LIN {X 0,Y 320.619,Z 422.638,A -85,B 0,C 180,E1 -15590.529,E2 -15590.529} C_VEL
LIN {X 0,Y 322.237,Z 412.256,A -85,B 0,C 180,E1 -15591.593,E2 -15591.593} C_VEL
LIN {X 0,Y 323.7,Z 399.843,A -85,B 0,C 180,E1 -15592.581,E2 -15592.581} C_VEL
LIN {X 0,Y 325.026,Z 386.792,A -85,B 0,C 180,E1 -15593.324,E2 -15593.324} C_VEL
LIN {X 0,Y 325.91,Z 373.737,A -85,B 0,C 180,E1 -15593.805,E2 -15593.805} C_VEL
LIN {X 0,Y 327.738,Z 306.835,A -85,B 0,C 180,E1 -15595.344,E2 -15595.344} C_VEL
LIN {X 0,Y 324.36,Z 288.516,A -85,B 0,C 180,E1 -15596.163,E2 -15596.163} C_VEL
LIN {X 0,Y 321.852,Z 278.173,A -85,B 0,C 180,E1 -15596.706,E2 -15596.706} C_VEL
LIN {X 0,Y 317.141,Z 267.501,A -85,B 0,C 180,E1 -15597.567,E2 -15597.567} C_VEL
LIN {X 0,Y 315.127,Z 258.496,A -85,B 0,C 180,E1 -15600.525,E2 -15600.525} C_VEL
LIN {X 0,Y 312.559,Z 248.178,A -85,B 0,C 180,E1 -15604.298,E2 -15604.298} C_VEL
LIN {X 0,Y 312.491,Z 248.049,A -85,B 0,C 180,E1 -15608.074,E2 -15608.074} C_VEL
LIN {X 0,Y 312.492,Z 248.056,A -85,B 0,C 180,E1 -15610.706,E2 -15610.706} C_VEL
LIN {X 0,Y 312.454,Z 248.066,A -85,B 0,C 180,E1 -15614.206,E2 -15614.206} C_VEL
LIN {X 0,Y 312.457,Z 248.052,A -85,B 0,C 180,E1 -15617.921,E2 -15617.921} C_VEL
LIN {X 0,Y 312.477,Z 248.06,A -85,B 0,C 180,E1 -15621.92,E2 -15621.92} C_VEL
LIN {X 0,Y 312.531,Z 248.049,A -85,B 0,C 180,E1 -15624.216,E2 -15624.216} C_VEL
LIN {X 0,Y 312.501,Z 248.051,A -85,B 0,C 180,E1 -15627.329,E2 -15627.329} C_VEL
LIN {X 0,Y 312.504,Z 248.052,A -85,B 0,C 180,E1 -15631.287,E2 -15631.287} C_VEL
LIN {X 0,Y 312.519,Z 248.048,A -85,B 0,C 180,E1 -15634.701,E2 -15634.701} C_VEL
LIN {X 0,Y 312.534,Z 248.051,A -85,B 0,C 180,E1 -15637.521,E2 -15637.521} C_VEL
LIN {X 0,Y 312.561,Z 248.048,A -85,B 0,C 180,E1 -15641.647,E2 -15641.647} C_VEL
LIN {X 0,Y 312.678,Z 248.036,A -85,B 0,C 180,E1 -15645.681,E2 -15645.681} C_VEL
LIN {X 0,Y 312.675,Z 248.038,A -85,B 0,C 180,E1 -15649.636,E2 -15649.636} C_VEL
LIN {X 0,Y 312.791,Z 248.009,A -85,B 0,C 180,E1 -15652.248,E2 -15652.248} C_VEL
LIN {X 0,Y 312.678,Z 248.036,A -85,B 0,C 180,E1 -15654.837,E2 -15654.837} C_VEL
LIN {X 0,Y 312.965,Z 247.999,A -85,B 0,C 180,E1 -15658.708,E2 -15658.708} C_VEL
LIN {X 0,Y 312.889,Z 248.007,A -85,B 0,C 180,E1 -15662.57,E2 -15662.57} C_VEL
LIN {X 0,Y 312.822,Z 248.015,A -85,B 0,C 180,E1 -15666.445,E2 -15666.445} C_VEL
LIN {X 0,Y 312.732,Z 248.024,A -85,B 0,C 180,E1 -15669.045,E2 -15669.045} C_VEL
LIN {X 0,Y 312.614,Z 248.037,A -85,B 0,C 180,E1 -15672.986,E2 -15672.986} C_VEL
LIN {X 0,Y 312.6,Z 248.046,A -85,B 0,C 180,E1 -15675.646,E2 -15675.646} C_VEL
LIN {X 0,Y 312.537,Z 248.05,A -85,B 0,C 180,E1 -15679.707,E2 -15679.707} C_VEL
LIN {X 0,Y 312.501,Z 248.054,A -85,B 0,C 180,E1 -15682.776,E2 -15682.776} C_VEL
LIN {X 0,Y 312.576,Z 248.047,A -85,B 0,C 180,E1 -15685.931,E2 -15685.931} C_VEL
LIN {X 0,Y 312.51,Z 248.047,A -85,B 0,C 180,E1 -15689.647,E2 -15689.647} C_VEL
LIN {X 0,Y 312.489,Z 248.056,A -85,B 0,C 180,E1 -15693.685,E2 -15693.685} C_VEL
LIN {X 0,Y 312.544,Z 248.146,A -85,B 0,C 180,E1 -15696.984,E2 -15696.984} C_VEL
LIN {X 0,Y 314.824,Z 257.191,A -85,B 0,C 180,E1 -15700.336,E2 -15700.336} C_VEL
LIN {X 0,Y 315.609,Z 260.248,A -85,B 0,C 180,E1 -15701.299,E2 -15701.299} C_VEL
LIN {X 0,Y 322.41,Z 274.835,A -85,B 0,C 180,E1 -15702.504,E2 -15702.504} C_VEL
LIN {X 0,Y 325.404,Z 282.157,A -85,B 0,C 180,E1 -15703.019,E2 -15703.019} C_VEL
LIN {X 0,Y 328.126,Z 295.692,A -85,B 0,C 180,E1 -15703.648,E2 -15703.648} C_VEL
LIN {X 0,Y 325.864,Z 368.46,A -85,B 0,C 180,E1 -15705.321,E2 -15705.321} C_VEL
LIN {X 0,Y 324.969,Z 381.92,A -85,B 0,C 180,E1 -15705.887,E2 -15705.887} C_VEL
LIN {X 0,Y 323.783,Z 394.274,A -85,B 0,C 180,E1 -15706.654,E2 -15706.654} C_VEL
LIN {X 0,Y 322.337,Z 406.019,A -85,B 0,C 180,E1 -15707.647,E2 -15707.647} C_VEL
LIN {X 0,Y 320.627,Z 417.406,A -85,B 0,C 180,E1 -15708.887,E2 -15708.887} C_VEL
LIN {X 0,Y 318.918,Z 427.555,A -85,B 0,C 180,E1 -15710.28,E2 -15710.28} C_VEL
LIN {X 0,Y 317.347,Z 435.854,A -85,B 0,C 180,E1 -15711.68,E2 -15711.68} C_VEL
LIN {X 0,Y 315.656,Z 444.602,A -85,B 0,C 180,E1 -15713.507,E2 -15713.507} C_VEL
LIN {X 0,Y 314.073,Z 452.692,A -85,B 0,C 180,E1 -15715.638,E2 -15715.638} C_VEL
LIN {X 0,Y 313.006,Z 457.984,A -85,B 0,C 180,E1 -15717.395,E2 -15717.395} C_VEL
LIN {X 0,Y 312.043,Z 463.111,A -85,B 0,C 180,E1 -15719.555,E2 -15719.555} C_VEL
LIN {X 0,Y 311.358,Z 466.861,A -85,B 0,C 180,E1 -15721.707,E2 -15721.707} C_VEL
LIN {X 0,Y 310.953,Z 468.664,A -85,B 0,C 180,E1 -15723.129,E2 -15723.129} C_VEL
LIN {X 0,Y 310.645,Z 470.184,A -85,B 0,C 180,E1 -15724.801,E2 -15724.801} C_VEL
LIN {X 0,Y 310.353,Z 471.184,A -85,B 0,C 180,E1 -15727.361,E2 -15727.361} C_VEL
LIN {X 0,Y 310.339,Z 471.111,A -85,B 0,C 180,E1 -15728.758,E2 -15728.758} C_VEL
LIN {X 0,Y 310.34,Z 470.552,A -85,B 0,C 180,E1 -15730.144,E2 -15730.144} C_VEL
LIN {X 0,Y 310.435,Z 469.179,A -85,B 0,C 180,E1 -15731.938,E2 -15731.938} C_VEL
LIN {X 0,Y 310.741,Z 466.186,A -85,B 0,C 180,E1 -15734.254,E2 -15734.254} C_VEL
LIN {X 0,Y 311.132,Z 462.559,A -85,B 0,C 180,E1 -15736.21,E2 -15736.21} C_VEL
LIN {X 0,Y 311.583,Z 457.45,A -85,B 0,C 180,E1 -15738.29,E2 -15738.29} C_VEL
LIN {X 0,Y 312.253,Z 451.179,A -85,B 0,C 180,E1 -15740.284,E2 -15740.284} C_VEL
LIN {X 0,Y 313.202,Z 443.354,A -85,B 0,C 180,E1 -15742.265,E2 -15742.265} C_VEL
LIN {X 0,Y 314.209,Z 435.298,A -85,B 0,C 180,E1 -15743.903,E2 -15743.903} C_VEL
LIN {X 0,Y 315.35,Z 425.459,A -85,B 0,C 180,E1 -15745.528,E2 -15745.528} C_VEL
LIN {X 0,Y 316.667,Z 414.664,A -85,B 0,C 180,E1 -15746.955,E2 -15746.955} C_VEL
LIN {X 0,Y 317.737,Z 403.761,A -85,B 0,C 180,E1 -15748.101,E2 -15748.101} C_VEL
LIN {X 0,Y 318.799,Z 390.855,A -85,B 0,C 180,E1 -15749.134,E2 -15749.134} C_VEL
LIN {X 0,Y 319.644,Z 377.868,A -85,B 0,C 180,E1 -15749.884,E2 -15749.884} C_VEL
LIN {X 0,Y 320.152,Z 365.22,A -85,B 0,C 180,E1 -15750.356,E2 -15750.356} C_VEL
LIN {X 0,Y 321.67,Z 292.026,A -85,B 0,C 180,E1 -15752.026,E2 -15752.026} C_VEL
LIN {X 0,Y 317.467,Z 267.45,A -85,B 0,C 180,E1 -15752.877,E2 -15752.877} C_VEL
LIN {X 0,Y 315.024,Z 260.027,A -85,B 0,C 180,E1 -15753.263,E2 -15753.263} C_VEL
LIN {X 0,Y 312.877,Z 248.346,A -85,B 0,C 180,E1 -15756.937,E2 -15756.937} C_VEL
LIN {X 0,Y 312.847,Z 248.014,A -85,B 0,C 180,E1 -15757.424,E2 -15757.424} C_VEL
LIN {X 0,Y 312.633,Z 248.042,A -85,B 0,C 180,E1 -15761.675,E2 -15761.675} C_VEL
LIN {X 0,Y 312.665,Z 248.034,A -85,B 0,C 180,E1 -15764.891,E2 -15764.891} C_VEL
LIN {X 0,Y 312.575,Z 248.047,A -85,B 0,C 180,E1 -15769.229,E2 -15769.229} C_VEL
LIN {X 0,Y 312.485,Z 248.057,A -85,B 0,C 180,E1 -15772.781,E2 -15772.781} C_VEL
LIN {X 0,Y 312.48,Z 248.062,A -85,B 0,C 180,E1 -15775.905,E2 -15775.905} C_VEL
LIN {X 0,Y 312.466,Z 248.062,A -85,B 0,C 180,E1 -15779.66,E2 -15779.66} C_VEL
LIN {X 0,Y 312.492,Z 248.055,A -85,B 0,C 180,E1 -15783.694,E2 -15783.694} C_VEL
LIN {X 0,Y 312.484,Z 248.057,A -85,B 0,C 180,E1 -15787.393,E2 -15787.393} C_VEL
LIN {X 0,Y 312.417,Z 248.067,A -85,B 0,C 180,E1 -15790.723,E2 -15790.723} C_VEL
LIN {X 0,Y 312.429,Z 248.066,A -85,B 0,C 180,E1 -15794.216,E2 -15794.216} C_VEL
LIN {X 0,Y 312.407,Z 248.064,A -85,B 0,C 180,E1 -15795.376,E2 -15795.376} C_VEL
LIN {X 0,Y 311.764,Z 248.149,A -85,B 0,C 180,E1 -15796.452,E2 -15796.452} C_VEL
LIN {X 0,Y 308.895,Z 248.501,A -85,B 0,C 180,E1 -15798.203,E2 -15798.203} C_VEL
LIN {X 0,Y 306.465,Z 248.801,A -85,B 0,C 180,E1 -15799.623,E2 -15799.623} C_VEL
LIN {X 0,Y 305.454,Z 248.931,A -85,B 0,C 180,E1 -15800.724,E2 -15800.724} C_VEL
LIN {X 0,Y 305.389,Z 248.936,A -85,B 0,C 180,E1 -15801.096,E2 -15801.096} C_VEL
LIN {X 0,Y 305.447,Z 248.939,A -85,B 0,C 180,E1 -15804.893,E2 -15804.893} C_VEL
LIN {X 0,Y 305.43,Z 248.932,A -85,B 0,C 180,E1 -15808.365,E2 -15808.365} C_VEL
LIN {X 0,Y 305.442,Z 248.928,A -85,B 0,C 180,E1 -15811.113,E2 -15811.113} C_VEL
LIN {X 0,Y 305.471,Z 248.93,A -85,B 0,C 180,E1 -15814.086,E2 -15814.086} C_VEL
LIN {X 0,Y 305.457,Z 248.932,A -85,B 0,C 180,E1 -15818.406,E2 -15818.406} C_VEL
LIN {X 0,Y 305.533,Z 248.912,A -85,B 0,C 180,E1 -15822.607,E2 -15822.607} C_VEL
LIN {X 0,Y 305.626,Z 248.906,A -85,B 0,C 180,E1 -15825.354,E2 -15825.354} C_VEL
LIN {X 0,Y 305.625,Z 248.913,A -85,B 0,C 180,E1 -15829.405,E2 -15829.405} C_VEL
LIN {X 0,Y 305.75,Z 248.898,A -85,B 0,C 180,E1 -15832.078,E2 -15832.078} C_VEL
LIN {X 0,Y 305.661,Z 248.9,A -85,B 0,C 180,E1 -15834.728,E2 -15834.728} C_VEL
LIN {X 0,Y 305.942,Z 248.868,A -85,B 0,C 180,E1 -15838.689,E2 -15838.689} C_VEL
LIN {X 0,Y 305.952,Z 248.87,A -85,B 0,C 180,E1 -15841.321,E2 -15841.321} C_VEL
LIN {X 0,Y 305.794,Z 248.889,A -85,B 0,C 180,E1 -15846.604,E2 -15846.604} C_VEL
LIN {X 0,Y 305.696,Z 248.892,A -85,B 0,C 180,E1 -15849.266,E2 -15849.266} C_VEL
LIN {X 0,Y 305.6,Z 248.915,A -85,B 0,C 180,E1 -15853.3,E2 -15853.3} C_VEL
LIN {X 0,Y 305.565,Z 248.92,A -85,B 0,C 180,E1 -15856.026,E2 -15856.026} C_VEL
LIN {X 0,Y 305.499,Z 248.921,A -85,B 0,C 180,E1 -15860.191,E2 -15860.191} C_VEL
LIN {X 0,Y 305.49,Z 248.93,A -85,B 0,C 180,E1 -15864.467,E2 -15864.467} C_VEL
LIN {X 0,Y 305.471,Z 248.931,A -85,B 0,C 180,E1 -15867.401,E2 -15867.401} C_VEL
LIN {X 0,Y 305.447,Z 248.929,A -85,B 0,C 180,E1 -15870.415,E2 -15870.415} C_VEL
LIN {X 0,Y 305.483,Z 248.93,A -85,B 0,C 180,E1 -15874.08,E2 -15874.08} C_VEL
LIN {X 0,Y 305.47,Z 248.928,A -85,B 0,C 180,E1 -15876.745,E2 -15876.745} C_VEL
LIN {X 0,Y 305.427,Z 248.937,A -85,B 0,C 180,E1 -15880.591,E2 -15880.591} C_VEL
LIN {X 0,Y 305.438,Z 248.938,A -85,B 0,C 180,E1 -15883.658,E2 -15883.658} C_VEL
LIN {X 0,Y 305.452,Z 248.935,A -85,B 0,C 180,E1 -15887.42,E2 -15887.42} C_VEL
LIN {X 0,Y 305.46,Z 248.933,A -85,B 0,C 180,E1 -15891.593,E2 -15891.593} C_VEL
LIN {X 0,Y 305.48,Z 248.929,A -85,B 0,C 180,E1 -15894.887,E2 -15894.887} C_VEL
LIN {X 0,Y 305.496,Z 248.932,A -85,B 0,C 180,E1 -15899.21,E2 -15899.21} C_VEL
LIN {X 0,Y 305.545,Z 249.228,A -85,B 0,C 180,E1 -15899.598,E2 -15899.598} C_VEL
LIN {X 0,Y 307.891,Z 260.415,A -85,B 0,C 180,E1 -15903.16,E2 -15903.16} C_VEL
LIN {X 0,Y 309.119,Z 267.787,A -85,B 0,C 180,E1 -15905.355,E2 -15905.355} C_VEL
LIN {X 0,Y 309.705,Z 271.988,A -85,B 0,C 180,E1 -15905.575,E2 -15905.575} C_VEL
LIN {X 0,Y 314.832,Z 306.06,A -85,B 0,C 180,E1 -15906.74,E2 -15906.74} C_VEL
LIN {X 0,Y 313.293,Z 375.551,A -85,B 0,C 180,E1 -15908.36,E2 -15908.36} C_VEL
LIN {X 0,Y 312.561,Z 388.819,A -85,B 0,C 180,E1 -15908.912,E2 -15908.912} C_VEL
LIN {X 0,Y 311.622,Z 401.603,A -85,B 0,C 180,E1 -15909.709,E2 -15909.709} C_VEL
LIN {X 0,Y 310.524,Z 412.959,A -85,B 0,C 180,E1 -15910.668,E2 -15910.668} C_VEL
LIN {X 0,Y 309.219,Z 424.684,A -85,B 0,C 180,E1 -15911.959,E2 -15911.959} C_VEL
LIN {X 0,Y 308.095,Z 434.783,A -85,B 0,C 180,E1 -15913.359,E2 -15913.359} C_VEL
LIN {X 0,Y 306.849,Z 444.708,A -85,B 0,C 180,E1 -15915.066,E2 -15915.066} C_VEL
LIN {X 0,Y 305.693,Z 453.833,A -85,B 0,C 180,E1 -15917.045,E2 -15917.045} C_VEL
LIN {X 0,Y 304.827,Z 461.173,A -85,B 0,C 180,E1 -15919.033,E2 -15919.033} C_VEL
LIN {X 0,Y 304.287,Z 466.122,A -85,B 0,C 180,E1 -15920.694,E2 -15920.694} C_VEL
LIN {X 0,Y 303.861,Z 470.917,A -85,B 0,C 180,E1 -15922.69,E2 -15922.69} C_VEL
LIN {X 0,Y 303.653,Z 474.574,A -85,B 0,C 180,E1 -15924.686,E2 -15924.686} C_VEL
LIN {X 0,Y 303.595,Z 476.458,A -85,B 0,C 180,E1 -15926.016,E2 -15926.016} C_VEL
LIN {X 0,Y 303.587,Z 477.869,A -85,B 0,C 180,E1 -15927.344,E2 -15927.344} C_VEL
LIN {X 0,Y 303.535,Z 478.867,A -85,B 0,C 180,E1 -15928.671,E2 -15928.671} C_VEL
LIN {X 0,Y 303.542,Z 479.476,A -85,B 0,C 180,E1 -15929.998,E2 -15929.998} C_VEL
LIN {X 0,Y 303.535,Z 479.694,A -85,B 0,C 180,E1 -15931.325,E2 -15931.325} C_VEL
LIN {X 0,Y 303.589,Z 479.483,A -85,B 0,C 180,E1 -15932.652,E2 -15932.652} C_VEL
LIN {X 0,Y 303.699,Z 477.887,A -85,B 0,C 180,E1 -15935.309,E2 -15935.309} C_VEL
LIN {X 0,Y 303.851,Z 476.507,A -85,B 0,C 180,E1 -15936.639,E2 -15936.639} C_VEL
LIN {X 0,Y 304.3,Z 473.604,A -85,B 0,C 180,E1 -15938.632,E2 -15938.632} C_VEL
LIN {X 0,Y 305,Z 469.69,A -85,B 0,C 180,E1 -15940.621,E2 -15940.621} C_VEL
LIN {X 0,Y 306.006,Z 464.664,A -85,B 0,C 180,E1 -15942.6,E2 -15942.6} C_VEL
LIN {X 0,Y 307.33,Z 458.369,A -85,B 0,C 180,E1 -15944.567,E2 -15944.567} C_VEL
LIN {X 0,Y 309.055,Z 450.506,A -85,B 0,C 180,E1 -15946.512,E2 -15946.512} C_VEL
LIN {X 0,Y 310.649,Z 441.952,A -85,B 0,C 180,E1 -15948.233,E2 -15948.233} C_VEL
LIN {X 0,Y 312.581,Z 431.757,A -85,B 0,C 180,E1 -15949.879,E2 -15949.879} C_VEL
LIN {X 0,Y 314.528,Z 420.616,A -85,B 0,C 180,E1 -15951.288,E2 -15951.288} C_VEL
LIN {X 0,Y 316.212,Z 409.737,A -85,B 0,C 180,E1 -15952.369,E2 -15952.369} C_VEL
LIN {X 0,Y 317.624,Z 397.768,A -85,B 0,C 180,E1 -15953.296,E2 -15953.296} C_VEL
LIN {X 0,Y 318.852,Z 385.459,A -85,B 0,C 180,E1 -15953.976,E2 -15953.976} C_VEL
LIN {X 0,Y 319.721,Z 372.89,A -85,B 0,C 180,E1 -15954.424,E2 -15954.424} C_VEL
LIN {X 0,Y 321.568,Z 307.683,A -85,B 0,C 180,E1 -15955.957,E2 -15955.957} C_VEL
LIN {X 0,Y 318.048,Z 288.778,A -85,B 0,C 180,E1 -15956.845,E2 -15956.845} C_VEL
LIN {X 0,Y 316.233,Z 281.362,A -85,B 0,C 180,E1 -15957.25,E2 -15957.25} C_VEL
LIN {X 0,Y 309.98,Z 267.54,A -85,B 0,C 180,E1 -15958.398,E2 -15958.398} C_VEL
LIN {X 0,Y 309.111,Z 263.636,A -85,B 0,C 180,E1 -15959.635,E2 -15959.635} C_VEL
LIN {X 0,Y 307.104,Z 255.27,A -85,B 0,C 180,E1 -15962.637,E2 -15962.637} C_VEL
LIN {X 0,Y 305.514,Z 249.002,A -85,B 0,C 180,E1 -15965.103,E2 -15965.103} C_VEL
LIN {X 0,Y 305.431,Z 248.928,A -85,B 0,C 180,E1 -15968.519,E2 -15968.519} C_VEL
LIN {X 0,Y 305.431,Z 248.924,A -85,B 0,C 180,E1 -15971.855,E2 -15971.855} C_VEL
LIN {X 0,Y 305.402,Z 248.93,A -85,B 0,C 180,E1 -15975.507,E2 -15975.507} C_VEL
LIN {X 0,Y 305.414,Z 248.932,A -85,B 0,C 180,E1 -15978.134,E2 -15978.134} C_VEL
LIN {X 0,Y 305.442,Z 248.936,A -85,B 0,C 180,E1 -15981.588,E2 -15981.588} C_VEL
LIN {X 0,Y 305.462,Z 248.935,A -85,B 0,C 180,E1 -15984.882,E2 -15984.882} C_VEL
LIN {X 0,Y 305.441,Z 248.935,A -85,B 0,C 180,E1 -15988.354,E2 -15988.354} C_VEL
LIN {X 0,Y 305.473,Z 248.927,A -85,B 0,C 180,E1 -15991.104,E2 -15991.104} C_VEL
LIN {X 0,Y 305.478,Z 248.928,A -85,B 0,C 180,E1 -15994.075,E2 -15994.075} C_VEL
LIN {X 0,Y 305.458,Z 248.928,A -85,B 0,C 180,E1 -15998.395,E2 -15998.395} C_VEL
LIN {X 0,Y 305.529,Z 248.92,A -85,B 0,C 180,E1 -16002.596,E2 -16002.596} C_VEL
LIN {X 0,Y 305.619,Z 248.917,A -85,B 0,C 180,E1 -16005.343,E2 -16005.343} C_VEL
LIN {X 0,Y 305.614,Z 248.915,A -85,B 0,C 180,E1 -16009.394,E2 -16009.394} C_VEL
LIN {X 0,Y 305.74,Z 248.888,A -85,B 0,C 180,E1 -16012.068,E2 -16012.068} C_VEL
LIN {X 0,Y 305.649,Z 248.911,A -85,B 0,C 180,E1 -16014.718,E2 -16014.718} C_VEL
LIN {X 0,Y 305.931,Z 248.875,A -85,B 0,C 180,E1 -16018.679,E2 -16018.679} C_VEL
LIN {X 0,Y 305.92,Z 248.869,A -85,B 0,C 180,E1 -16021.311,E2 -16021.311} C_VEL
LIN {X 0,Y 305.641,Z 248.905,A -85,B 0,C 180,E1 -16025.272,E2 -16025.272} C_VEL
LIN {X 0,Y 305.728,Z 248.902,A -85,B 0,C 180,E1 -16027.922,E2 -16027.922} C_VEL
LIN {X 0,Y 305.579,Z 248.92,A -85,B 0,C 180,E1 -16031.94,E2 -16031.94} C_VEL
LIN {X 0,Y 305.588,Z 248.919,A -85,B 0,C 180,E1 -16035.009,E2 -16035.009} C_VEL
LIN {X 0,Y 305.519,Z 248.924,A -85,B 0,C 180,E1 -16039.422,E2 -16039.422} C_VEL
LIN {X 0,Y 305.461,Z 248.932,A -85,B 0,C 180,E1 -16043.035,E2 -16043.035} C_VEL
LIN {X 0,Y 305.52,Z 248.929,A -85,B 0,C 180,E1 -16046.222,E2 -16046.222} C_VEL
LIN {X 0,Y 305.46,Z 248.92,A -85,B 0,C 180,E1 -16049.043,E2 -16049.043} C_VEL
LIN {X 0,Y 305.413,Z 248.932,A -85,B 0,C 180,E1 -16051.948,E2 -16051.948} C_VEL
LIN {X 0,Y 305.484,Z 249.005,A -85,B 0,C 180,E1 -16056.206,E2 -16056.206} C_VEL
LIN {X 0,Y 307.819,Z 258.157,A -85,B 0,C 180,E1 -16059.73,E2 -16059.73} C_VEL
LIN {X 0,Y 308.403,Z 260.428,A -85,B 0,C 180,E1 -16060.439,E2 -16060.439} C_VEL
LIN {X 0,Y 314.332,Z 272.513,A -85,B 0,C 180,E1 -16061.526,E2 -16061.526} C_VEL
LIN {X 0,Y 319.535,Z 284.486,A -85,B 0,C 180,E1 -16062.442,E2 -16062.442} C_VEL
LIN {X 0,Y 321.983,Z 297,A -85,B 0,C 180,E1 -16063.042,E2 -16063.042} C_VEL
LIN {X 0,Y 319.664,Z 368.312,A -85,B 0,C 180,E1 -16064.714,E2 -16064.714} C_VEL
LIN {X 0,Y 318.791,Z 381.04,A -85,B 0,C 180,E1 -16065.248,E2 -16065.248} C_VEL
LIN {X 0,Y 317.528,Z 393.61,A -85,B 0,C 180,E1 -16066.021,E2 -16066.021} C_VEL
LIN {X 0,Y 316.09,Z 405.087,A -85,B 0,C 180,E1 -16066.983,E2 -16066.983} C_VEL
LIN {X 0,Y 314.228,Z 417.05,A -85,B 0,C 180,E1 -16068.291,E2 -16068.291} C_VEL
LIN {X 0,Y 312.416,Z 427.335,A -85,B 0,C 180,E1 -16069.717,E2 -16069.717} C_VEL
LIN {X 0,Y 310.769,Z 435.634,A -85,B 0,C 180,E1 -16071.133,E2 -16071.133} C_VEL
LIN {X 0,Y 308.931,Z 444.73,A -85,B 0,C 180,E1 -16073.062,E2 -16073.062} C_VEL
LIN {X 0,Y 307.298,Z 452.462,A -85,B 0,C 180,E1 -16075.13,E2 -16075.13} C_VEL
LIN {X 0,Y 305.951,Z 458.903,A -85,B 0,C 180,E1 -16077.331,E2 -16077.331} C_VEL
LIN {X 0,Y 304.951,Z 463.792,A -85,B 0,C 180,E1 -16079.537,E2 -16079.537} C_VEL
LIN {X 0,Y 304.382,Z 466.801,A -85,B 0,C 180,E1 -16081.315,E2 -16081.315} C_VEL
LIN {X 0,Y 303.707,Z 469.752,A -85,B 0,C 180,E1 -16083.92,E2 -16083.92} C_VEL
LIN {X 0,Y 303.474,Z 470.741,A -85,B 0,C 180,E1 -16085.366,E2 -16085.366} C_VEL
LIN {X 0,Y 303.261,Z 471.3,A -85,B 0,C 180,E1 -16087.951,E2 -16087.951} C_VEL
LIN {X 0,Y 303.22,Z 470.862,A -85,B 0,C 180,E1 -16089.658,E2 -16089.658} C_VEL
LIN {X 0,Y 303.319,Z 469.386,A -85,B 0,C 180,E1 -16091.779,E2 -16091.779} C_VEL
LIN {X 0,Y 303.686,Z 465.807,A -85,B 0,C 180,E1 -16094.568,E2 -16094.568} C_VEL
LIN {X 0,Y 304.108,Z 461.865,A -85,B 0,C 180,E1 -16096.64,E2 -16096.64} C_VEL
LIN {X 0,Y 304.622,Z 456.742,A -85,B 0,C 180,E1 -16098.693,E2 -16098.693} C_VEL
LIN {X 0,Y 305.369,Z 450.28,A -85,B 0,C 180,E1 -16100.731,E2 -16100.731} C_VEL
LIN {X 0,Y 306.38,Z 442.144,A -85,B 0,C 180,E1 -16102.754,E2 -16102.754} C_VEL
LIN {X 0,Y 307.427,Z 433.829,A -85,B 0,C 180,E1 -16104.427,E2 -16104.427} C_VEL
LIN {X 0,Y 308.7,Z 423.659,A -85,B 0,C 180,E1 -16106.086,E2 -16106.086} C_VEL
LIN {X 0,Y 309.898,Z 413.559,A -85,B 0,C 180,E1 -16107.402,E2 -16107.402} C_VEL
LIN {X 0,Y 311.012,Z 402.562,A -85,B 0,C 180,E1 -16108.545,E2 -16108.545} C_VEL
LIN {X 0,Y 312.019,Z 390.453,A -85,B 0,C 180,E1 -16109.518,E2 -16109.518} C_VEL
LIN {X 0,Y 312.834,Z 378.084,A -85,B 0,C 180,E1 -16110.243,E2 -16110.243} C_VEL
LIN {X 0,Y 313.35,Z 365.555,A -85,B 0,C 180,E1 -16110.725,E2 -16110.725} C_VEL
LIN {X 0,Y 314.878,Z 292.515,A -85,B 0,C 180,E1 -16112.43,E2 -16112.43} C_VEL
LIN {X 0,Y 311.028,Z 269.782,A -85,B 0,C 180,E1 -16113.233,E2 -16113.233} C_VEL
LIN {X 0,Y 307.869,Z 260.473,A -85,B 0,C 180,E1 -16113.707,E2 -16113.707} C_VEL
LIN {X 0,Y 307.408,Z 258.332,A -85,B 0,C 180,E1 -16114.263,E2 -16114.263} C_VEL
LIN {X 0,Y 305.847,Z 249.195,A -85,B 0,C 180,E1 -16117.263,E2 -16117.263} C_VEL
LIN {X 0,Y 305.759,Z 248.899,A -85,B 0,C 180,E1 -16117.929,E2 -16117.929} C_VEL
LIN {X 0,Y 305.567,Z 248.921,A -85,B 0,C 180,E1 -16121.948,E2 -16121.948} C_VEL
LIN {X 0,Y 305.603,Z 248.915,A -85,B 0,C 180,E1 -16125.038,E2 -16125.038} C_VEL
LIN {X 0,Y 305.545,Z 248.921,A -85,B 0,C 180,E1 -16128.787,E2 -16128.787} C_VEL
LIN {X 0,Y 305.439,Z 248.935,A -85,B 0,C 180,E1 -16133.037,E2 -16133.037} C_VEL
LIN {X 0,Y 305.424,Z 248.939,A -85,B 0,C 180,E1 -16136.196,E2 -16136.196} C_VEL
LIN {X 0,Y 305.418,Z 248.939,A -85,B 0,C 180,E1 -16139.038,E2 -16139.038} C_VEL
LIN {X 0,Y 305.407,Z 248.941,A -85,B 0,C 180,E1 -16141.958,E2 -16141.958} C_VEL
LIN {X 0,Y 305.434,Z 248.936,A -85,B 0,C 180,E1 -16145.119,E2 -16145.119} C_VEL
LIN {X 0,Y 305.41,Z 248.939,A -85,B 0,C 180,E1 -16148.53,E2 -16148.53} C_VEL
LIN {X 0,Y 305.412,Z 248.942,A -85,B 0,C 180,E1 -16152.587,E2 -16152.587} C_VEL
LIN {X 0,Y 305.401,Z 248.941,A -85,B 0,C 180,E1 -16156.35,E2 -16156.35} C_VEL
LIN {X 0,Y 305.393,Z 248.934,A -85,B 0,C 180,E1 -16159.891,E2 -16159.891} C_VEL
LIN {X 0,Y 305.389,Z 248.936,A -85,B 0,C 180,E1 -16161.096,E2 -16161.096} C_VEL
LIN {X 0,Y 304.761,Z 249.02,A -85,B 0,C 180,E1 -16162.197,E2 -16162.197} C_VEL
LIN {X 0,Y 301.896,Z 249.376,A -85,B 0,C 180,E1 -16163.987,E2 -16163.987} C_VEL
LIN {X 0,Y 299.458,Z 249.681,A -85,B 0,C 180,E1 -16165.44,E2 -16165.44} C_VEL
LIN {X 0,Y 298.435,Z 249.808,A -85,B 0,C 180,E1 -16166.566,E2 -16166.566} C_VEL
LIN {X 0,Y 298.367,Z 249.813,A -85,B 0,C 180,E1 -16166.948,E2 -16166.948} C_VEL
LIN {X 0,Y 298.354,Z 249.806,A -85,B 0,C 180,E1 -16170.645,E2 -16170.645} C_VEL
LIN {X 0,Y 298.41,Z 249.811,A -85,B 0,C 180,E1 -16174.924,E2 -16174.924} C_VEL
LIN {X 0,Y 298.388,Z 249.814,A -85,B 0,C 180,E1 -16177.868,E2 -16177.868} C_VEL
LIN {X 0,Y 298.46,Z 249.799,A -85,B 0,C 180,E1 -16180.758,E2 -16180.758} C_VEL
LIN {X 0,Y 298.586,Z 249.78,A -85,B 0,C 180,E1 -16185,E2 -16185} C_VEL
LIN {X 0,Y 298.584,Z 249.789,A -85,B 0,C 180,E1 -16189.152,E2 -16189.152} C_VEL
LIN {X 0,Y 298.701,Z 249.777,A -85,B 0,C 180,E1 -16191.89,E2 -16191.89} C_VEL
LIN {X 0,Y 298.631,Z 249.775,A -85,B 0,C 180,E1 -16194.604,E2 -16194.604} C_VEL
LIN {X 0,Y 298.91,Z 249.744,A -85,B 0,C 180,E1 -16198.658,E2 -16198.658} C_VEL
LIN {X 0,Y 298.918,Z 249.746,A -85,B 0,C 180,E1 -16201.352,E2 -16201.352} C_VEL
LIN {X 0,Y 298.743,Z 249.766,A -85,B 0,C 180,E1 -16206.76,E2 -16206.76} C_VEL
LIN {X 0,Y 298.629,Z 249.77,A -85,B 0,C 180,E1 -16209.487,E2 -16209.487} C_VEL
LIN {X 0,Y 298.559,Z 249.791,A -85,B 0,C 180,E1 -16213.62,E2 -16213.62} C_VEL
LIN {X 0,Y 298.499,Z 249.803,A -85,B 0,C 180,E1 -16216.416,E2 -16216.416} C_VEL
LIN {X 0,Y 298.461,Z 249.797,A -85,B 0,C 180,E1 -16219.622,E2 -16219.622} C_VEL
LIN {X 0,Y 298.437,Z 249.807,A -85,B 0,C 180,E1 -16223.604,E2 -16223.604} C_VEL
LIN {X 0,Y 298.424,Z 249.811,A -85,B 0,C 180,E1 -16226.585,E2 -16226.585} C_VEL
LIN {X 0,Y 298.41,Z 249.806,A -85,B 0,C 180,E1 -16229.647,E2 -16229.647} C_VEL
LIN {X 0,Y 298.411,Z 249.812,A -85,B 0,C 180,E1 -16232.803,E2 -16232.803} C_VEL
LIN {X 0,Y 298.444,Z 249.803,A -85,B 0,C 180,E1 -16236.804,E2 -16236.804} C_VEL
LIN {X 0,Y 298.365,Z 249.82,A -85,B 0,C 180,E1 -16241.27,E2 -16241.27} C_VEL
LIN {X 0,Y 298.374,Z 249.817,A -85,B 0,C 180,E1 -16245.036,E2 -16245.036} C_VEL
LIN {X 0,Y 298.365,Z 249.817,A -85,B 0,C 180,E1 -16248.923,E2 -16248.923} C_VEL
LIN {X 0,Y 298.405,Z 249.811,A -85,B 0,C 180,E1 -16252.238,E2 -16252.238} C_VEL
LIN {X 0,Y 298.426,Z 249.809,A -85,B 0,C 180,E1 -16255.581,E2 -16255.581} C_VEL
LIN {X 0,Y 298.482,Z 249.977,A -85,B 0,C 180,E1 -16259.193,E2 -16259.193} C_VEL
LIN {X 0,Y 300.666,Z 260.544,A -85,B 0,C 180,E1 -16262.66,E2 -16262.66} C_VEL
LIN {X 0,Y 301.982,Z 267.843,A -85,B 0,C 180,E1 -16264.888,E2 -16264.888} C_VEL
LIN {X 0,Y 302.909,Z 271.921,A -85,B 0,C 180,E1 -16265.107,E2 -16265.107} C_VEL
LIN {X 0,Y 308.143,Z 307.18,A -85,B 0,C 180,E1 -16266.344,E2 -16266.344} C_VEL
LIN {X 0,Y 306.506,Z 375.971,A -85,B 0,C 180,E1 -16267.989,E2 -16267.989} C_VEL
LIN {X 0,Y 305.707,Z 389.831,A -85,B 0,C 180,E1 -16268.593,E2 -16268.593} C_VEL
LIN {X 0,Y 304.752,Z 402.31,A -85,B 0,C 180,E1 -16269.408,E2 -16269.408} C_VEL
LIN {X 0,Y 303.61,Z 413.44,A -85,B 0,C 180,E1 -16270.386,E2 -16270.386} C_VEL
LIN {X 0,Y 302.268,Z 425.059,A -85,B 0,C 180,E1 -16271.704,E2 -16271.704} C_VEL
LIN {X 0,Y 301.125,Z 435.026,A -85,B 0,C 180,E1 -16273.129,E2 -16273.129} C_VEL
LIN {X 0,Y 299.968,Z 444.073,A -85,B 0,C 180,E1 -16274.716,E2 -16274.716} C_VEL
LIN {X 0,Y 298.744,Z 453.301,A -85,B 0,C 180,E1 -16276.738,E2 -16276.738} C_VEL
LIN {X 0,Y 297.819,Z 460.717,A -85,B 0,C 180,E1 -16278.772,E2 -16278.772} C_VEL
LIN {X 0,Y 297.258,Z 465.735,A -85,B 0,C 180,E1 -16280.472,E2 -16280.472} C_VEL
LIN {X 0,Y 296.807,Z 470.592,A -85,B 0,C 180,E1 -16282.515,E2 -16282.515} C_VEL
LIN {X 0,Y 296.568,Z 474.306,A -85,B 0,C 180,E1 -16284.559,E2 -16284.559} C_VEL
LIN {X 0,Y 296.498,Z 476.22,A -85,B 0,C 180,E1 -16285.92,E2 -16285.92} C_VEL
LIN {X 0,Y 296.492,Z 477.681,A -85,B 0,C 180,E1 -16287.281,E2 -16287.281} C_VEL
LIN {X 0,Y 296.457,Z 478.706,A -85,B 0,C 180,E1 -16288.639,E2 -16288.639} C_VEL
LIN {X 0,Y 296.46,Z 479.34,A -85,B 0,C 180,E1 -16289.998,E2 -16289.998} C_VEL
LIN {X 0,Y 296.457,Z 479.586,A -85,B 0,C 180,E1 -16291.356,E2 -16291.356} C_VEL
LIN {X 0,Y 296.495,Z 479.421,A -85,B 0,C 180,E1 -16292.715,E2 -16292.715} C_VEL
LIN {X 0,Y 296.614,Z 477.876,A -85,B 0,C 180,E1 -16295.436,E2 -16295.436} C_VEL
LIN {X 0,Y 296.774,Z 476.522,A -85,B 0,C 180,E1 -16296.798,E2 -16296.798} C_VEL
LIN {X 0,Y 297.283,Z 473.671,A -85,B 0,C 180,E1 -16298.837,E2 -16298.837} C_VEL
LIN {X 0,Y 298.009,Z 469.812,A -85,B 0,C 180,E1 -16300.873,E2 -16300.873} C_VEL
LIN {X 0,Y 299.061,Z 464.845,A -85,B 0,C 180,E1 -16302.898,E2 -16302.898} C_VEL
LIN {X 0,Y 300.465,Z 458.623,A -85,B 0,C 180,E1 -16304.907,E2 -16304.907} C_VEL
LIN {X 0,Y 302.274,Z 450.863,A -85,B 0,C 180,E1 -16306.893,E2 -16306.893} C_VEL
LIN {X 0,Y 303.891,Z 442.669,A -85,B 0,C 180,E1 -16308.601,E2 -16308.601} C_VEL
LIN {X 0,Y 305.755,Z 433.401,A -85,B 0,C 180,E1 -16310.166,E2 -16310.166} C_VEL
LIN {X 0,Y 307.705,Z 422.794,A -85,B 0,C 180,E1 -16311.608,E2 -16311.608} C_VEL
LIN {X 0,Y 309.462,Z 412.535,A -85,B 0,C 180,E1 -16312.708,E2 -16312.708} C_VEL
LIN {X 0,Y 311.054,Z 400.329,A -85,B 0,C 180,E1 -16313.73,E2 -16313.73} C_VEL
LIN {X 0,Y 312.475,Z 387.547,A -85,B 0,C 180,E1 -16314.497,E2 -16314.497} C_VEL
LIN {X 0,Y 313.411,Z 375.296,A -85,B 0,C 180,E1 -16314.994,E2 -16314.994} C_VEL
LIN {X 0,Y 315.544,Z 309.217,A -85,B 0,C 180,E1 -16316.574,E2 -16316.574} C_VEL
LIN {X 0,Y 312.147,Z 290.747,A -85,B 0,C 180,E1 -16317.466,E2 -16317.466} C_VEL
LIN {X 0,Y 310.492,Z 284.171,A -85,B 0,C 180,E1 -16317.843,E2 -16317.843} C_VEL
LIN {X 0,Y 304.299,Z 270.733,A -85,B 0,C 180,E1 -16318.989,E2 -16318.989} C_VEL
LIN {X 0,Y 302.698,Z 267.125,A -85,B 0,C 180,E1 -16319.367,E2 -16319.367} C_VEL
LIN {X 0,Y 300.526,Z 257.979,A -85,B 0,C 180,E1 -16322.654,E2 -16322.654} C_VEL
LIN {X 0,Y 298.485,Z 249.854,A -85,B 0,C 180,E1 -16325.933,E2 -16325.933} C_VEL
LIN {X 0,Y 298.401,Z 249.811,A -85,B 0,C 180,E1 -16329.484,E2 -16329.484} C_VEL
LIN {X 0,Y 298.404,Z 249.804,A -85,B 0,C 180,E1 -16333.099,E2 -16333.099} C_VEL
LIN {X 0,Y 298.373,Z 249.797,A -85,B 0,C 180,E1 -16336.91,E2 -16336.91} C_VEL
LIN {X 0,Y 298.386,Z 249.812,A -85,B 0,C 180,E1 -16341.006,E2 -16341.006} C_VEL
LIN {X 0,Y 298.405,Z 249.808,A -85,B 0,C 180,E1 -16343.923,E2 -16343.923} C_VEL
LIN {X 0,Y 298.392,Z 249.808,A -85,B 0,C 180,E1 -16347.195,E2 -16347.195} C_VEL
LIN {X 0,Y 298.4,Z 249.808,A -85,B 0,C 180,E1 -16350.62,E2 -16350.62} C_VEL
LIN {X 0,Y 298.419,Z 249.804,A -85,B 0,C 180,E1 -16354.913,E2 -16354.913} C_VEL
LIN {X 0,Y 298.413,Z 249.804,A -85,B 0,C 180,E1 -16359.308,E2 -16359.308} C_VEL
LIN {X 0,Y 298.46,Z 249.804,A -85,B 0,C 180,E1 -16362.17,E2 -16362.17} C_VEL
LIN {X 0,Y 298.579,Z 249.791,A -85,B 0,C 180,E1 -16364.989,E2 -16364.989} C_VEL
LIN {X 0,Y 298.573,Z 249.788,A -85,B 0,C 180,E1 -16369.141,E2 -16369.141} C_VEL
LIN {X 0,Y 298.691,Z 249.767,A -85,B 0,C 180,E1 -16371.879,E2 -16371.879} C_VEL
LIN {X 0,Y 298.619,Z 249.786,A -85,B 0,C 180,E1 -16374.593,E2 -16374.593} C_VEL
LIN {X 0,Y 298.898,Z 249.751,A -85,B 0,C 180,E1 -16378.648,E2 -16378.648} C_VEL
LIN {X 0,Y 298.888,Z 249.744,A -85,B 0,C 180,E1 -16381.342,E2 -16381.342} C_VEL
LIN {X 0,Y 298.716,Z 249.773,A -85,B 0,C 180,E1 -16386.75,E2 -16386.75} C_VEL
LIN {X 0,Y 298.607,Z 249.781,A -85,B 0,C 180,E1 -16389.477,E2 -16389.477} C_VEL
LIN {X 0,Y 298.525,Z 249.792,A -85,B 0,C 180,E1 -16393.611,E2 -16393.611} C_VEL
LIN {X 0,Y 298.464,Z 249.8,A -85,B 0,C 180,E1 -16396.407,E2 -16396.407} C_VEL
LIN {X 0,Y 298.46,Z 249.803,A -85,B 0,C 180,E1 -16399.634,E2 -16399.634} C_VEL
LIN {X 0,Y 298.404,Z 249.813,A -85,B 0,C 180,E1 -16403.595,E2 -16403.595} C_VEL
LIN {X 0,Y 298.463,Z 249.809,A -85,B 0,C 180,E1 -16406.57,E2 -16406.57} C_VEL
LIN {X 0,Y 298.388,Z 249.805,A -85,B 0,C 180,E1 -16409.637,E2 -16409.637} C_VEL
LIN {X 0,Y 298.365,Z 249.807,A -85,B 0,C 180,E1 -16412.796,E2 -16412.796} C_VEL
LIN {X 0,Y 298.451,Z 250.001,A -85,B 0,C 180,E1 -16415.486,E2 -16415.486} C_VEL
LIN {X 0,Y 300.973,Z 259.754,A -85,B 0,C 180,E1 -16419.308,E2 -16419.308} C_VEL
LIN {X 0,Y 301.279,Z 260.736,A -85,B 0,C 180,E1 -16419.541,E2 -16419.541} C_VEL
LIN {X 0,Y 307.689,Z 273.459,A -85,B 0,C 180,E1 -16420.753,E2 -16420.753} C_VEL
LIN {X 0,Y 313.686,Z 286.953,A -85,B 0,C 180,E1 -16421.845,E2 -16421.845} C_VEL
LIN {X 0,Y 315.871,Z 297.519,A -85,B 0,C 180,E1 -16422.383,E2 -16422.383} C_VEL
LIN {X 0,Y 313.496,Z 368.122,A -85,B 0,C 180,E1 -16424.066,E2 -16424.066} C_VEL
LIN {X 0,Y 312.594,Z 381.26,A -85,B 0,C 180,E1 -16424.628,E2 -16424.628} C_VEL
LIN {X 0,Y 311.356,Z 393.171,A -85,B 0,C 180,E1 -16425.371,E2 -16425.371} C_VEL
LIN {X 0,Y 309.878,Z 404.362,A -85,B 0,C 180,E1 -16426.305,E2 -16426.305} C_VEL
LIN {X 0,Y 308.124,Z 415.346,A -85,B 0,C 180,E1 -16427.494,E2 -16427.494} C_VEL
LIN {X 0,Y 306.205,Z 425.87,A -85,B 0,C 180,E1 -16428.935,E2 -16428.935} C_VEL
LIN {X 0,Y 304.235,Z 435.432,A -85,B 0,C 180,E1 -16430.563,E2 -16430.563} C_VEL
LIN {X 0,Y 302.342,Z 444.314,A -85,B 0,C 180,E1 -16432.461,E2 -16432.461} C_VEL
LIN {X 0,Y 300.515,Z 452.526,A -85,B 0,C 180,E1 -16434.69,E2 -16434.69} C_VEL
LIN {X 0,Y 299.3,Z 457.857,A -85,B 0,C 180,E1 -16436.511,E2 -16436.511} C_VEL
LIN {X 0,Y 298.174,Z 463.06,A -85,B 0,C 180,E1 -16438.768,E2 -16438.768} C_VEL
LIN {X 0,Y 297.421,Z 466.788,A -85,B 0,C 180,E1 -16440.948,E2 -16440.948} C_VEL
LIN {X 0,Y 296.756,Z 469.502,A -85,B 0,C 180,E1 -16443.261,E2 -16443.261} C_VEL
LIN {X 0,Y 296.456,Z 470.593,A -85,B 0,C 180,E1 -16444.743,E2 -16444.743} C_VEL
LIN {X 0,Y 296.253,Z 471.241,A -85,B 0,C 180,E1 -16446.219,E2 -16446.219} C_VEL
LIN {X 0,Y 296.171,Z 471.412,A -85,B 0,C 180,E1 -16447.717,E2 -16447.717} C_VEL
LIN {X 0,Y 296.138,Z 471.112,A -85,B 0,C 180,E1 -16449.149,E2 -16449.149} C_VEL
LIN {X 0,Y 296.234,Z 469.603,A -85,B 0,C 180,E1 -16451.595,E2 -16451.595} C_VEL
LIN {X 0,Y 296.524,Z 466.549,A -85,B 0,C 180,E1 -16454.185,E2 -16454.185} C_VEL
LIN {X 0,Y 296.946,Z 462.813,A -85,B 0,C 180,E1 -16456.312,E2 -16456.312} C_VEL
LIN {X 0,Y 297.442,Z 457.913,A -85,B 0,C 180,E1 -16458.416,E2 -16458.416} C_VEL
LIN {X 0,Y 298.118,Z 451.709,A -85,B 0,C 180,E1 -16460.504,E2 -16460.504} C_VEL
LIN {X 0,Y 299.114,Z 443.961,A -85,B 0,C 180,E1 -16462.577,E2 -16462.577} C_VEL
LIN {X 0,Y 300.213,Z 436.003,A -85,B 0,C 180,E1 -16464.292,E2 -16464.292} C_VEL
LIN {X 0,Y 301.435,Z 426.268,A -85,B 0,C 180,E1 -16465.991,E2 -16465.991} C_VEL
LIN {X 0,Y 302.849,Z 415.385,A -85,B 0,C 180,E1 -16467.508,E2 -16467.508} C_VEL
LIN {X 0,Y 303.922,Z 404.921,A -85,B 0,C 180,E1 -16468.677,E2 -16468.677} C_VEL
LIN {X 0,Y 305.032,Z 392.37,A -85,B 0,C 180,E1 -16469.755,E2 -16469.755} C_VEL
LIN {X 0,Y 306.012,Z 379.051,A -85,B 0,C 180,E1 -16470.578,E2 -16470.578} C_VEL
LIN {X 0,Y 306.566,Z 365.882,A -85,B 0,C 180,E1 -16471.11,E2 -16471.11} C_VEL
LIN {X 0,Y 308.242,Z 293.769,A -85,B 0,C 180,E1 -16472.821,E2 -16472.821} C_VEL
LIN {X 0,Y 304.529,Z 271.9,A -85,B 0,C 180,E1 -16473.615,E2 -16473.615} C_VEL
LIN {X 0,Y 300.66,Z 260.596,A -85,B 0,C 180,E1 -16474.212,E2 -16474.212} C_VEL
LIN {X 0,Y 300.266,Z 258.66,A -85,B 0,C 180,E1 -16474.701,E2 -16474.701} C_VEL
LIN {X 0,Y 298.778,Z 249.894,A -85,B 0,C 180,E1 -16477.69,E2 -16477.69} C_VEL
LIN {X 0,Y 298.518,Z 249.798,A -85,B 0,C 180,E1 -16482.235,E2 -16482.235} C_VEL
LIN {X 0,Y 298.551,Z 249.793,A -85,B 0,C 180,E1 -16485.198,E2 -16485.198} C_VEL
LIN {X 0,Y 298.491,Z 249.801,A -85,B 0,C 180,E1 -16489.248,E2 -16489.248} C_VEL
LIN {X 0,Y 298.379,Z 249.817,A -85,B 0,C 180,E1 -16493.606,E2 -16493.606} C_VEL
LIN {X 0,Y 298.373,Z 249.815,A -85,B 0,C 180,E1 -16496.588,E2 -16496.588} C_VEL
LIN {X 0,Y 298.364,Z 249.819,A -85,B 0,C 180,E1 -16499.649,E2 -16499.649} C_VEL
LIN {X 0,Y 298.365,Z 249.814,A -85,B 0,C 180,E1 -16502.806,E2 -16502.806} C_VEL
LIN {X 0,Y 298.377,Z 249.818,A -85,B 0,C 180,E1 -16506.078,E2 -16506.078} C_VEL
LIN {X 0,Y 298.35,Z 249.812,A -85,B 0,C 180,E1 -16509.498,E2 -16509.498} C_VEL
LIN {X 0,Y 298.348,Z 249.82,A -85,B 0,C 180,E1 -16513.103,E2 -16513.103} C_VEL
LIN {X 0,Y 298.351,Z 249.816,A -85,B 0,C 180,E1 -16516.921,E2 -16516.921} C_VEL
LIN {X 0,Y 298.365,Z 249.815,A -85,B 0,C 180,E1 -16521.087,E2 -16521.087} C_VEL
LIN {X 0,Y 298.39,Z 249.813,A -85,B 0,C 180,E1 -16523.934,E2 -16523.934} C_VEL
LIN {X 0,Y 298.367,Z 249.813,A -85,B 0,C 180,E1 -16526.948,E2 -16526.948} C_VEL
LIN {X 0,Y 297.731,Z 249.896,A -85,B 0,C 180,E1 -16528.075,E2 -16528.075} C_VEL
LIN {X 0,Y 294.866,Z 250.248,A -85,B 0,C 180,E1 -16529.909,E2 -16529.909} C_VEL
LIN {X 0,Y 292.426,Z 250.549,A -85,B 0,C 180,E1 -16531.398,E2 -16531.398} C_VEL
LIN {X 0,Y 291.397,Z 250.678,A -85,B 0,C 180,E1 -16532.552,E2 -16532.552} C_VEL
LIN {X 0,Y 291.324,Z 250.689,A -85,B 0,C 180,E1 -16532.943,E2 -16532.943} C_VEL
LIN {X 0,Y 291.345,Z 250.695,A -85,B 0,C 180,E1 -16537.303,E2 -16537.303} C_VEL
LIN {X 0,Y 291.384,Z 250.68,A -85,B 0,C 180,E1 -16540.271,E2 -16540.271} C_VEL
LIN {X 0,Y 291.498,Z 250.661,A -85,B 0,C 180,E1 -16544.672,E2 -16544.672} C_VEL
LIN {X 0,Y 291.53,Z 250.667,A -85,B 0,C 180,E1 -16548.886,E2 -16548.886} C_VEL
LIN {X 0,Y 291.655,Z 250.655,A -85,B 0,C 180,E1 -16551.693,E2 -16551.693} C_VEL
LIN {X 0,Y 291.601,Z 250.65,A -85,B 0,C 180,E1 -16554.473,E2 -16554.473} C_VEL
LIN {X 0,Y 291.877,Z 250.619,A -85,B 0,C 180,E1 -16558.626,E2 -16558.626} C_VEL
LIN {X 0,Y 291.885,Z 250.622,A -85,B 0,C 180,E1 -16561.385,E2 -16561.385} C_VEL
LIN {X 0,Y 291.694,Z 250.642,A -85,B 0,C 180,E1 -16566.924,E2 -16566.924} C_VEL
LIN {X 0,Y 291.575,Z 250.647,A -85,B 0,C 180,E1 -16569.719,E2 -16569.719} C_VEL
LIN {X 0,Y 291.529,Z 250.667,A -85,B 0,C 180,E1 -16573.955,E2 -16573.955} C_VEL
LIN {X 0,Y 291.443,Z 250.681,A -85,B 0,C 180,E1 -16576.825,E2 -16576.825} C_VEL
LIN {X 0,Y 291.407,Z 250.674,A -85,B 0,C 180,E1 -16579.846,E2 -16579.846} C_VEL
LIN {X 0,Y 291.375,Z 250.687,A -85,B 0,C 180,E1 -16584.212,E2 -16584.212} C_VEL
LIN {X 0,Y 291.369,Z 250.688,A -85,B 0,C 180,E1 -16587.282,E2 -16587.282} C_VEL
LIN {X 0,Y 291.336,Z 250.686,A -85,B 0,C 180,E1 -16590.442,E2 -16590.442} C_VEL
LIN {X 0,Y 291.362,Z 250.69,A -85,B 0,C 180,E1 -16593.701,E2 -16593.701} C_VEL
LIN {X 0,Y 291.371,Z 250.686,A -85,B 0,C 180,E1 -16597.25,E2 -16597.25} C_VEL
LIN {X 0,Y 291.313,Z 250.695,A -85,B 0,C 180,E1 -16601.59,E2 -16601.59} C_VEL
LIN {X 0,Y 291.301,Z 250.701,A -85,B 0,C 180,E1 -16605.598,E2 -16605.598} C_VEL
LIN {X 0,Y 291.318,Z 250.697,A -85,B 0,C 180,E1 -16609.353,E2 -16609.353} C_VEL
LIN {X 0,Y 291.404,Z 250.683,A -85,B 0,C 180,E1 -16612.917,E2 -16612.917} C_VEL
LIN {X 0,Y 291.362,Z 250.69,A -85,B 0,C 180,E1 -16616.302,E2 -16616.302} C_VEL
LIN {X 0,Y 291.4,Z 250.758,A -85,B 0,C 180,E1 -16618.764,E2 -16618.764} C_VEL
LIN {X 0,Y 292.493,Z 255.757,A -85,B 0,C 180,E1 -16620.54,E2 -16620.54} C_VEL
LIN {X 0,Y 294.411,Z 265.765,A -85,B 0,C 180,E1 -16623.791,E2 -16623.791} C_VEL
LIN {X 0,Y 294.844,Z 267.983,A -85,B 0,C 180,E1 -16624.397,E2 -16624.397} C_VEL
LIN {X 0,Y 296.433,Z 273.898,A -85,B 0,C 180,E1 -16624.692,E2 -16624.692} C_VEL
LIN {X 0,Y 301.388,Z 307.184,A -85,B 0,C 180,E1 -16625.9,E2 -16625.9} C_VEL
LIN {X 0,Y 299.723,Z 376.385,A -85,B 0,C 180,E1 -16627.6,E2 -16627.6} C_VEL
LIN {X 0,Y 298.912,Z 390.078,A -85,B 0,C 180,E1 -16628.218,E2 -16628.218} C_VEL
LIN {X 0,Y 297.865,Z 402.946,A -85,B 0,C 180,E1 -16629.09,E2 -16629.09} C_VEL
LIN {X 0,Y 296.523,Z 415.515,A -85,B 0,C 180,E1 -16630.258,E2 -16630.258} C_VEL
LIN {X 0,Y 295.145,Z 426.73,A -85,B 0,C 180,E1 -16631.606,E2 -16631.606} C_VEL
LIN {X 0,Y 293.97,Z 437.018,A -85,B 0,C 180,E1 -16633.183,E2 -16633.183} C_VEL
LIN {X 0,Y 292.582,Z 446.756,A -85,B 0,C 180,E1 -16635.033,E2 -16635.033} C_VEL
LIN {X 0,Y 291.604,Z 454.137,A -85,B 0,C 180,E1 -16636.762,E2 -16636.762} C_VEL
LIN {X 0,Y 290.689,Z 461.384,A -85,B 0,C 180,E1 -16638.846,E2 -16638.846} C_VEL
LIN {X 0,Y 290.043,Z 467.143,A -85,B 0,C 180,E1 -16640.936,E2 -16640.936} C_VEL
LIN {X 0,Y 289.652,Z 471.663,A -85,B 0,C 180,E1 -16643.03,E2 -16643.03} C_VEL
LIN {X 0,Y 289.492,Z 474.169,A -85,B 0,C 180,E1 -16644.51,E2 -16644.51} C_VEL
LIN {X 0,Y 289.4,Z 477.491,A -85,B 0,C 180,E1 -16647.214,E2 -16647.214} C_VEL
LIN {X 0,Y 289.381,Z 478.544,A -85,B 0,C 180,E1 -16648.606,E2 -16648.606} C_VEL
LIN {X 0,Y 289.381,Z 479.203,A -85,B 0,C 180,E1 -16649.998,E2 -16649.998} C_VEL
LIN {X 0,Y 289.38,Z 479.475,A -85,B 0,C 180,E1 -16651.389,E2 -16651.389} C_VEL
LIN {X 0,Y 289.403,Z 479.354,A -85,B 0,C 180,E1 -16652.782,E2 -16652.782} C_VEL
LIN {X 0,Y 289.531,Z 477.864,A -85,B 0,C 180,E1 -16655.57,E2 -16655.57} C_VEL
LIN {X 0,Y 289.726,Z 476.536,A -85,B 0,C 180,E1 -16656.964,E2 -16656.964} C_VEL
LIN {X 0,Y 290.254,Z 473.738,A -85,B 0,C 180,E1 -16659.053,E2 -16659.053} C_VEL
LIN {X 0,Y 291.011,Z 469.934,A -85,B 0,C 180,E1 -16661.137,E2 -16661.137} C_VEL
LIN {X 0,Y 292.135,Z 465.034,A -85,B 0,C 180,E1 -16663.209,E2 -16663.209} C_VEL
LIN {X 0,Y 293.618,Z 458.893,A -85,B 0,C 180,E1 -16665.263,E2 -16665.263} C_VEL
LIN {X 0,Y 295.504,Z 451.271,A -85,B 0,C 180,E1 -16667.292,E2 -16667.292} C_VEL
LIN {X 0,Y 297.165,Z 443.357,A -85,B 0,C 180,E1 -16669.006,E2 -16669.006} C_VEL
LIN {X 0,Y 299.134,Z 434.056,A -85,B 0,C 180,E1 -16670.633,E2 -16670.633} C_VEL
LIN {X 0,Y 301.162,Z 423.602,A -85,B 0,C 180,E1 -16672.102,E2 -16672.102} C_VEL
LIN {X 0,Y 303.253,Z 411.957,A -85,B 0,C 180,E1 -16673.381,E2 -16673.381} C_VEL
LIN {X 0,Y 304.942,Z 399.574,A -85,B 0,C 180,E1 -16674.416,E2 -16674.416} C_VEL
LIN {X 0,Y 306.392,Z 386.578,A -85,B 0,C 180,E1 -16675.198,E2 -16675.198} C_VEL
LIN {X 0,Y 307.385,Z 373.662,A -85,B 0,C 180,E1 -16675.7,E2 -16675.7} C_VEL
LIN {X 0,Y 309.444,Z 309.932,A -85,B 0,C 180,E1 -16677.25,E2 -16677.25} C_VEL
LIN {X 0,Y 305.72,Z 289.825,A -85,B 0,C 180,E1 -16678.261,E2 -16678.261} C_VEL
LIN {X 0,Y 304.309,Z 285.795,A -85,B 0,C 180,E1 -16678.552,E2 -16678.552} C_VEL
LIN {X 0,Y 298.663,Z 273.683,A -85,B 0,C 180,E1 -16679.641,E2 -16679.641} C_VEL
LIN {X 0,Y 295.516,Z 267.137,A -85,B 0,C 180,E1 -16680.321,E2 -16680.321} C_VEL
LIN {X 0,Y 294.344,Z 262.324,A -85,B 0,C 180,E1 -16682.045,E2 -16682.045} C_VEL
LIN {X 0,Y 292.056,Z 253.144,A -85,B 0,C 180,E1 -16685.698,E2 -16685.698} C_VEL
LIN {X 0,Y 291.41,Z 250.714,A -85,B 0,C 180,E1 -16686.834,E2 -16686.834} C_VEL
LIN {X 0,Y 291.331,Z 250.691,A -85,B 0,C 180,E1 -16690.639,E2 -16690.639} C_VEL
LIN {X 0,Y 291.296,Z 250.701,A -85,B 0,C 180,E1 -16694.397,E2 -16694.397} C_VEL
LIN {X 0,Y 291.297,Z 250.693,A -85,B 0,C 180,E1 -16698.407,E2 -16698.407} C_VEL
LIN {X 0,Y 291.334,Z 250.691,A -85,B 0,C 180,E1 -16701.15,E2 -16701.15} C_VEL
LIN {X 0,Y 291.355,Z 250.689,A -85,B 0,C 180,E1 -16704.62,E2 -16704.62} C_VEL
LIN {X 0,Y 291.365,Z 250.686,A -85,B 0,C 180,E1 -16707.945,E2 -16707.945} C_VEL
LIN {X 0,Y 291.341,Z 250.687,A -85,B 0,C 180,E1 -16711.149,E2 -16711.149} C_VEL
LIN {X 0,Y 291.344,Z 250.687,A -85,B 0,C 180,E1 -16714.26,E2 -16714.26} C_VEL
LIN {X 0,Y 291.347,Z 250.692,A -85,B 0,C 180,E1 -16717.292,E2 -16717.292} C_VEL
LIN {X 0,Y 291.384,Z 250.685,A -85,B 0,C 180,E1 -16720.26,E2 -16720.26} C_VEL
LIN {X 0,Y 291.491,Z 250.671,A -85,B 0,C 180,E1 -16724.66,E2 -16724.66} C_VEL
LIN {X 0,Y 291.52,Z 250.665,A -85,B 0,C 180,E1 -16728.875,E2 -16728.875} C_VEL
LIN {X 0,Y 291.644,Z 250.645,A -85,B 0,C 180,E1 -16731.682,E2 -16731.682} C_VEL
LIN {X 0,Y 291.589,Z 250.662,A -85,B 0,C 180,E1 -16734.462,E2 -16734.462} C_VEL
LIN {X 0,Y 291.864,Z 250.627,A -85,B 0,C 180,E1 -16738.615,E2 -16738.615} C_VEL
LIN {X 0,Y 291.856,Z 250.62,A -85,B 0,C 180,E1 -16741.374,E2 -16741.374} C_VEL
LIN {X 0,Y 291.668,Z 250.651,A -85,B 0,C 180,E1 -16746.914,E2 -16746.914} C_VEL
LIN {X 0,Y 291.55,Z 250.66,A -85,B 0,C 180,E1 -16749.709,E2 -16749.709} C_VEL
LIN {X 0,Y 291.495,Z 250.67,A -85,B 0,C 180,E1 -16753.946,E2 -16753.946} C_VEL
LIN {X 0,Y 291.418,Z 250.678,A -85,B 0,C 180,E1 -16756.816,E2 -16756.816} C_VEL
LIN {X 0,Y 291.401,Z 250.682,A -85,B 0,C 180,E1 -16759.855,E2 -16759.855} C_VEL
LIN {X 0,Y 291.358,Z 250.693,A -85,B 0,C 180,E1 -16764.202,E2 -16764.202} C_VEL
LIN {X 0,Y 291.394,Z 250.682,A -85,B 0,C 180,E1 -16767.267,E2 -16767.267} C_VEL
LIN {X 0,Y 291.306,Z 250.698,A -85,B 0,C 180,E1 -16770.433,E2 -16770.433} C_VEL
LIN {X 0,Y 291.367,Z 250.798,A -85,B 0,C 180,E1 -16774.555,E2 -16774.555} C_VEL
LIN {X 0,Y 293.42,Z 258.493,A -85,B 0,C 180,E1 -16777.78,E2 -16777.78} C_VEL
LIN {X 0,Y 294.036,Z 260.72,A -85,B 0,C 180,E1 -16778.523,E2 -16778.523} C_VEL
LIN {X 0,Y 302.022,Z 276.249,A -85,B 0,C 180,E1 -16780.119,E2 -16780.119} C_VEL
LIN {X 0,Y 308.162,Z 290.262,A -85,B 0,C 180,E1 -16781.285,E2 -16781.285} C_VEL
LIN {X 0,Y 309.801,Z 298.456,A -85,B 0,C 180,E1 -16781.71,E2 -16781.71} C_VEL
LIN {X 0,Y 307.373,Z 368.474,A -85,B 0,C 180,E1 -16783.416,E2 -16783.416} C_VEL
LIN {X 0,Y 306.394,Z 381.696,A -85,B 0,C 180,E1 -16783.993,E2 -16783.993} C_VEL
LIN {X 0,Y 305.071,Z 393.979,A -85,B 0,C 180,E1 -16784.782,E2 -16784.782} C_VEL
LIN {X 0,Y 303.455,Z 405.495,A -85,B 0,C 180,E1 -16785.785,E2 -16785.785} C_VEL
LIN {X 0,Y 301.579,Z 416.556,A -85,B 0,C 180,E1 -16787.031,E2 -16787.031} C_VEL
LIN {X 0,Y 299.598,Z 426.773,A -85,B 0,C 180,E1 -16788.48,E2 -16788.48} C_VEL
LIN {X 0,Y 297.738,Z 435.302,A -85,B 0,C 180,E1 -16789.97,E2 -16789.97} C_VEL
LIN {X 0,Y 295.76,Z 444.003,A -85,B 0,C 180,E1 -16791.846,E2 -16791.846} C_VEL
LIN {X 0,Y 293.927,Z 451.833,A -85,B 0,C 180,E1 -16793.985,E2 -16793.985} C_VEL
LIN {X 0,Y 292.249,Z 458.803,A -85,B 0,C 180,E1 -16796.423,E2 -16796.423} C_VEL
LIN {X 0,Y 291.087,Z 463.77,A -85,B 0,C 180,E1 -16798.731,E2 -16798.731} C_VEL
LIN {X 0,Y 290.277,Z 467.415,A -85,B 0,C 180,E1 -16801.041,E2 -16801.041} C_VEL
LIN {X 0,Y 289.823,Z 469.172,A -85,B 0,C 180,E1 -16802.568,E2 -16802.568} C_VEL
LIN {X 0,Y 289.496,Z 470.445,A -85,B 0,C 180,E1 -16804.091,E2 -16804.091} C_VEL
LIN {X 0,Y 289.216,Z 471.194,A -85,B 0,C 180,E1 -16805.603,E2 -16805.603} C_VEL
LIN {X 0,Y 289.082,Z 471.524,A -85,B 0,C 180,E1 -16807.474,E2 -16807.474} C_VEL
LIN {X 0,Y 289.029,Z 470.732,A -85,B 0,C 180,E1 -16810.1,E2 -16810.1} C_VEL
LIN {X 0,Y 289.131,Z 469.676,A -85,B 0,C 180,E1 -16811.582,E2 -16811.582} C_VEL
LIN {X 0,Y 289.367,Z 467.227,A -85,B 0,C 180,E1 -16813.784,E2 -16813.784} C_VEL
LIN {X 0,Y 289.77,Z 463.711,A -85,B 0,C 180,E1 -16815.966,E2 -16815.966} C_VEL
LIN {X 0,Y 290.251,Z 459.061,A -85,B 0,C 180,E1 -16818.125,E2 -16818.125} C_VEL
LIN {X 0,Y 290.924,Z 453.123,A -85,B 0,C 180,E1 -16820.267,E2 -16820.267} C_VEL
LIN {X 0,Y 291.885,Z 445.655,A -85,B 0,C 180,E1 -16822.392,E2 -16822.392} C_VEL
LIN {X 0,Y 293.225,Z 436.344,A -85,B 0,C 180,E1 -16824.501,E2 -16824.501} C_VEL
LIN {X 0,Y 294.463,Z 426.681,A -85,B 0,C 180,E1 -16826.239,E2 -16826.239} C_VEL
LIN {X 0,Y 295.899,Z 416.021,A -85,B 0,C 180,E1 -16827.77,E2 -16827.77} C_VEL
LIN {X 0,Y 297.038,Z 405.473,A -85,B 0,C 180,E1 -16828.985,E2 -16828.985} C_VEL
LIN {X 0,Y 298.183,Z 393.113,A -85,B 0,C 180,E1 -16830.087,E2 -16830.087} C_VEL
LIN {X 0,Y 299.186,Z 380.021,A -85,B 0,C 180,E1 -16830.927,E2 -16830.927} C_VEL
LIN {X 0,Y 299.756,Z 367.535,A -85,B 0,C 180,E1 -16831.472,E2 -16831.472} C_VEL
LIN {X 0,Y 301.462,Z 294.226,A -85,B 0,C 180,E1 -16833.258,E2 -16833.258} C_VEL
LIN {X 0,Y 298.018,Z 273.813,A -85,B 0,C 180,E1 -16834.021,E2 -16834.021} C_VEL
LIN {X 0,Y 293.481,Z 260.659,A -85,B 0,C 180,E1 -16834.737,E2 -16834.737} C_VEL
LIN {X 0,Y 293.319,Z 259.912,A -85,B 0,C 180,E1 -16834.882,E2 -16834.882} C_VEL
LIN {X 0,Y 291.731,Z 250.904,A -85,B 0,C 180,E1 -16837.964,E2 -16837.964} C_VEL
LIN {X 0,Y 291.651,Z 250.654,A -85,B 0,C 180,E1 -16838.938,E2 -16838.938} C_VEL
LIN {X 0,Y 291.486,Z 250.676,A -85,B 0,C 180,E1 -16843.954,E2 -16843.954} C_VEL
LIN {X 0,Y 291.452,Z 250.667,A -85,B 0,C 180,E1 -16846.822,E2 -16846.822} C_VEL
LIN {X 0,Y 291.419,Z 250.687,A -85,B 0,C 180,E1 -16849.879,E2 -16849.879} C_VEL
LIN {X 0,Y 291.317,Z 250.699,A -85,B 0,C 180,E1 -16854.215,E2 -16854.215} C_VEL
LIN {X 0,Y 291.305,Z 250.694,A -85,B 0,C 180,E1 -16857.286,E2 -16857.286} C_VEL
LIN {X 0,Y 291.289,Z 250.7,A -85,B 0,C 180,E1 -16860.445,E2 -16860.445} C_VEL
LIN {X 0,Y 291.316,Z 250.691,A -85,B 0,C 180,E1 -16863.704,E2 -16863.704} C_VEL
LIN {X 0,Y 291.327,Z 250.692,A -85,B 0,C 180,E1 -16867.253,E2 -16867.253} C_VEL
LIN {X 0,Y 291.277,Z 250.697,A -85,B 0,C 180,E1 -16870.654,E2 -16870.654} C_VEL
LIN {X 0,Y 291.262,Z 250.704,A -85,B 0,C 180,E1 -16874.41,E2 -16874.41} C_VEL
LIN {X 0,Y 291.277,Z 250.695,A -85,B 0,C 180,E1 -16878.418,E2 -16878.418} C_VEL
LIN {X 0,Y 291.318,Z 250.695,A -85,B 0,C 180,E1 -16881.162,E2 -16881.162} C_VEL
LIN {X 0,Y 291.341,Z 250.694,A -85,B 0,C 180,E1 -16884.631,E2 -16884.631} C_VEL
LIN {X 0,Y 291.354,Z 250.684,A -85,B 0,C 180,E1 -16887.956,E2 -16887.956} C_VEL
LIN {X 0,Y 291.305,Z 250.686,A -85,B 0,C 180,E1 -16891.157,E2 -16891.157} C_VEL
LIN {X 0,Y 291.324,Z 250.689,A -85,B 0,C 180,E1 -16892.943,E2 -16892.943} C_VEL
LIN {X 0,Y 290.679,Z 250.775,A -85,B 0,C 180,E1 -16894.097,E2 -16894.097} C_VEL
LIN {X 0,Y 287.817,Z 251.133,A -85,B 0,C 180,E1 -16895.977,E2 -16895.977} C_VEL
LIN {X 0,Y 285.385,Z 251.437,A -85,B 0,C 180,E1 -16897.503,E2 -16897.503} C_VEL
LIN {X 0,Y 284.358,Z 251.56,A -85,B 0,C 180,E1 -16898.686,E2 -16898.686} C_VEL
LIN {X 0,Y 284.284,Z 251.565,A -85,B 0,C 180,E1 -16899.086,E2 -16899.086} C_VEL
LIN {X 0,Y 284.367,Z 251.544,A -85,B 0,C 180,E1 -16902.754,E2 -16902.754} C_VEL
LIN {X 0,Y 284.463,Z 251.542,A -85,B 0,C 180,E1 -16905.703,E2 -16905.703} C_VEL
LIN {X 0,Y 284.517,Z 251.544,A -85,B 0,C 180,E1 -16910.049,E2 -16910.049} C_VEL
LIN {X 0,Y 284.645,Z 251.521,A -85,B 0,C 180,E1 -16912.914,E2 -16912.914} C_VEL
LIN {X 0,Y 284.844,Z 251.495,A -85,B 0,C 180,E1 -16918.592,E2 -16918.592} C_VEL
LIN {X 0,Y 284.851,Z 251.498,A -85,B 0,C 180,E1 -16921.419,E2 -16921.419} C_VEL
LIN {X 0,Y 284.647,Z 251.518,A -85,B 0,C 180,E1 -16927.097,E2 -16927.097} C_VEL
LIN {X 0,Y 284.523,Z 251.525,A -85,B 0,C 180,E1 -16929.962,E2 -16929.962} C_VEL
LIN {X 0,Y 284.477,Z 251.548,A -85,B 0,C 180,E1 -16934.308,E2 -16934.308} C_VEL
LIN {X 0,Y 284.348,Z 251.558,A -85,B 0,C 180,E1 -16938.747,E2 -16938.747} C_VEL
LIN {X 0,Y 284.343,Z 251.564,A -85,B 0,C 180,E1 -16943.3,E2 -16943.3} C_VEL
LIN {X 0,Y 284.346,Z 251.563,A -85,B 0,C 180,E1 -16947.149,E2 -16947.149} C_VEL
LIN {X 0,Y 284.313,Z 251.56,A -85,B 0,C 180,E1 -16950.094,E2 -16950.094} C_VEL
LIN {X 0,Y 284.323,Z 251.568,A -85,B 0,C 180,E1 -16952.948,E2 -16952.948} C_VEL
LIN {X 0,Y 284.337,Z 251.558,A -85,B 0,C 180,E1 -16956.39,E2 -16956.39} C_VEL
LIN {X 0,Y 284.274,Z 251.573,A -85,B 0,C 180,E1 -16960.005,E2 -16960.005} C_VEL
LIN {X 0,Y 284.252,Z 251.576,A -85,B 0,C 180,E1 -16964.189,E2 -16964.189} C_VEL
LIN {X 0,Y 284.257,Z 251.577,A -85,B 0,C 180,E1 -16968.119,E2 -16968.119} C_VEL
LIN {X 0,Y 284.314,Z 251.564,A -85,B 0,C 180,E1 -16971.829,E2 -16971.829} C_VEL
LIN {X 0,Y 284.326,Z 251.564,A -85,B 0,C 180,E1 -16975.351,E2 -16975.351} C_VEL
LIN {X 0,Y 284.359,Z 251.674,A -85,B 0,C 180,E1 -16978.42,E2 -16978.42} C_VEL
LIN {X 0,Y 286.103,Z 260.067,A -85,B 0,C 180,E1 -16981.378,E2 -16981.378} C_VEL
LIN {X 0,Y 287.569,Z 267.634,A -85,B 0,C 180,E1 -16983.815,E2 -16983.815} C_VEL
LIN {X 0,Y 289.639,Z 274.055,A -85,B 0,C 180,E1 -16984.203,E2 -16984.203} C_VEL
LIN {X 0,Y 294.726,Z 308.622,A -85,B 0,C 180,E1 -16985.479,E2 -16985.479} C_VEL
LIN {X 0,Y 293.016,Z 375.635,A -85,B 0,C 180,E1 -16987.152,E2 -16987.152} C_VEL
LIN {X 0,Y 292.173,Z 389.542,A -85,B 0,C 180,E1 -16987.782,E2 -16987.782} C_VEL
LIN {X 0,Y 291.176,Z 401.498,A -85,B 0,C 180,E1 -16988.586,E2 -16988.586} C_VEL
LIN {X 0,Y 290.031,Z 412.813,A -85,B 0,C 180,E1 -16989.613,E2 -16989.613} C_VEL
LIN {X 0,Y 288.656,Z 423.191,A -85,B 0,C 180,E1 -16990.809,E2 -16990.809} C_VEL
LIN {X 0,Y 287.333,Z 434.381,A -85,B 0,C 180,E1 -16992.451,E2 -16992.451} C_VEL
LIN {X 0,Y 285.96,Z 444.491,A -85,B 0,C 180,E1 -16994.313,E2 -16994.313} C_VEL
LIN {X 0,Y 284.66,Z 453.604,A -85,B 0,C 180,E1 -16996.433,E2 -16996.433} C_VEL
LIN {X 0,Y 283.68,Z 460.933,A -85,B 0,C 180,E1 -16998.566,E2 -16998.566} C_VEL
LIN {X 0,Y 282.991,Z 466.78,A -85,B 0,C 180,E1 -17000.708,E2 -17000.708} C_VEL
LIN {X 0,Y 282.588,Z 471.365,A -85,B 0,C 180,E1 -17002.855,E2 -17002.855} C_VEL
LIN {X 0,Y 282.41,Z 474.179,A -85,B 0,C 180,E1 -17004.557,E2 -17004.557} C_VEL
LIN {X 0,Y 282.31,Z 477.288,A -85,B 0,C 180,E1 -17007.144,E2 -17007.144} C_VEL
LIN {X 0,Y 282.306,Z 478.382,A -85,B 0,C 180,E1 -17008.571,E2 -17008.571} C_VEL
LIN {X 0,Y 282.304,Z 479.066,A -85,B 0,C 180,E1 -17009.998,E2 -17009.998} C_VEL
LIN {X 0,Y 282.305,Z 479.363,A -85,B 0,C 180,E1 -17011.424,E2 -17011.424} C_VEL
LIN {X 0,Y 282.314,Z 479.275,A -85,B 0,C 180,E1 -17012.852,E2 -17012.852} C_VEL
LIN {X 0,Y 282.438,Z 478.019,A -85,B 0,C 180,E1 -17015.503,E2 -17015.503} C_VEL
LIN {X 0,Y 282.675,Z 476.556,A -85,B 0,C 180,E1 -17017.139,E2 -17017.139} C_VEL
LIN {X 0,Y 283.238,Z 473.82,A -85,B 0,C 180,E1 -17019.279,E2 -17019.279} C_VEL
LIN {X 0,Y 284.025,Z 470.087,A -85,B 0,C 180,E1 -17021.415,E2 -17021.415} C_VEL
LIN {X 0,Y 285.201,Z 465.259,A -85,B 0,C 180,E1 -17023.536,E2 -17023.536} C_VEL
LIN {X 0,Y 286.789,Z 459.191,A -85,B 0,C 180,E1 -17025.636,E2 -17025.636} C_VEL
LIN {X 0,Y 288.747,Z 451.668,A -85,B 0,C 180,E1 -17027.71,E2 -17027.71} C_VEL
LIN {X 0,Y 290.441,Z 444.061,A -85,B 0,C 180,E1 -17029.421,E2 -17029.421} C_VEL
LIN {X 0,Y 292.551,Z 434.708,A -85,B 0,C 180,E1 -17031.119,E2 -17031.119} C_VEL
LIN {X 0,Y 294.649,Z 424.409,A -85,B 0,C 180,E1 -17032.617,E2 -17032.617} C_VEL
LIN {X 0,Y 296.796,Z 412.992,A -85,B 0,C 180,E1 -17033.921,E2 -17033.921} C_VEL
LIN {X 0,Y 298.557,Z 401.05,A -85,B 0,C 180,E1 -17034.974,E2 -17034.974} C_VEL
LIN {X 0,Y 300.145,Z 387.842,A -85,B 0,C 180,E1 -17035.807,E2 -17035.807} C_VEL
LIN {X 0,Y 301.233,Z 374.652,A -85,B 0,C 180,E1 -17036.36,E2 -17036.36} C_VEL
LIN {X 0,Y 303.432,Z 310.958,A -85,B 0,C 180,E1 -17037.939,E2 -17037.939} C_VEL
LIN {X 0,Y 299.915,Z 291.798,A -85,B 0,C 180,E1 -17038.938,E2 -17038.938} C_VEL
LIN {X 0,Y 294.358,Z 279.12,A -85,B 0,C 180,E1 -17040.07,E2 -17040.07} C_VEL
LIN {X 0,Y 288.274,Z 266.962,A -85,B 0,C 180,E1 -17041.376,E2 -17041.376} C_VEL
LIN {X 0,Y 285.804,Z 256.929,A -85,B 0,C 180,E1 -17045.334,E2 -17045.334} C_VEL
LIN {X 0,Y 284.312,Z 251.597,A -85,B 0,C 180,E1 -17047.77,E2 -17047.77} C_VEL
LIN {X 0,Y 284.311,Z 251.572,A -85,B 0,C 180,E1 -17049.99,E2 -17049.99} C_VEL
LIN {X 0,Y 284.251,Z 251.579,A -85,B 0,C 180,E1 -17054.186,E2 -17054.186} C_VEL
LIN {X 0,Y 284.242,Z 251.567,A -85,B 0,C 180,E1 -17058.114,E2 -17058.114} C_VEL
LIN {X 0,Y 284.297,Z 251.571,A -85,B 0,C 180,E1 -17061.823,E2 -17061.823} C_VEL
LIN {X 0,Y 284.307,Z 251.571,A -85,B 0,C 180,E1 -17065.345,E2 -17065.345} C_VEL
LIN {X 0,Y 284.284,Z 251.574,A -85,B 0,C 180,E1 -17068.719,E2 -17068.719} C_VEL
LIN {X 0,Y 284.279,Z 251.571,A -85,B 0,C 180,E1 -17071.979,E2 -17071.979} C_VEL
LIN {X 0,Y 284.294,Z 251.569,A -85,B 0,C 180,E1 -17076.152,E2 -17076.152} C_VEL
LIN {X 0,Y 284.329,Z 251.562,A -85,B 0,C 180,E1 -17079.923,E2 -17079.923} C_VEL
LIN {X 0,Y 284.44,Z 251.548,A -85,B 0,C 180,E1 -17084.488,E2 -17084.488} C_VEL
LIN {X 0,Y 284.473,Z 251.541,A -85,B 0,C 180,E1 -17088.596,E2 -17088.596} C_VEL
LIN {X 0,Y 284.601,Z 251.524,A -85,B 0,C 180,E1 -17091.474,E2 -17091.474} C_VEL
LIN {X 0,Y 284.559,Z 251.538,A -85,B 0,C 180,E1 -17094.325,E2 -17094.325} C_VEL
LIN {X 0,Y 284.83,Z 251.503,A -85,B 0,C 180,E1 -17098.581,E2 -17098.581} C_VEL
LIN {X 0,Y 284.823,Z 251.496,A -85,B 0,C 180,E1 -17101.408,E2 -17101.408} C_VEL
LIN {X 0,Y 284.624,Z 251.529,A -85,B 0,C 180,E1 -17107.086,E2 -17107.086} C_VEL
LIN {X 0,Y 284.496,Z 251.539,A -85,B 0,C 180,E1 -17109.952,E2 -17109.952} C_VEL
LIN {X 0,Y 284.443,Z 251.551,A -85,B 0,C 180,E1 -17114.299,E2 -17114.299} C_VEL
LIN {X 0,Y 284.352,Z 251.564,A -85,B 0,C 180,E1 -17118.735,E2 -17118.735} C_VEL
LIN {X 0,Y 284.291,Z 251.572,A -85,B 0,C 180,E1 -17121.759,E2 -17121.759} C_VEL
LIN {X 0,Y 284.313,Z 251.566,A -85,B 0,C 180,E1 -17124.842,E2 -17124.842} C_VEL
LIN {X 0,Y 284.301,Z 251.557,A -85,B 0,C 180,E1 -17128.006,E2 -17128.006} C_VEL
LIN {X 0,Y 284.265,Z 251.572,A -85,B 0,C 180,E1 -17131.27,E2 -17131.27} C_VEL
LIN {X 0,Y 284.296,Z 251.631,A -85,B 0,C 180,E1 -17133.574,E2 -17133.574} C_VEL
LIN {X 0,Y 285.879,Z 257.353,A -85,B 0,C 180,E1 -17136.149,E2 -17136.149} C_VEL
LIN {X 0,Y 286.788,Z 260.748,A -85,B 0,C 180,E1 -17137.44,E2 -17137.44} C_VEL
LIN {X 0,Y 293.53,Z 273.431,A -85,B 0,C 180,E1 -17138.876,E2 -17138.876} C_VEL
LIN {X 0,Y 299.96,Z 286.926,A -85,B 0,C 180,E1 -17140.161,E2 -17140.161} C_VEL
LIN {X 0,Y 302.704,Z 293.954,A -85,B 0,C 180,E1 -17140.72,E2 -17140.72} C_VEL
LIN {X 0,Y 303.816,Z 299.764,A -85,B 0,C 180,E1 -17141.025,E2 -17141.025} C_VEL
LIN {X 0,Y 301.302,Z 368.254,A -85,B 0,C 180,E1 -17142.715,E2 -17142.715} C_VEL
LIN {X 0,Y 300.283,Z 381.667,A -85,B 0,C 180,E1 -17143.308,E2 -17143.308} C_VEL
LIN {X 0,Y 298.957,Z 393.518,A -85,B 0,C 180,E1 -17144.075,E2 -17144.075} C_VEL
LIN {X 0,Y 297.354,Z 404.667,A -85,B 0,C 180,E1 -17145.04,E2 -17145.04} C_VEL
LIN {X 0,Y 295.303,Z 416.327,A -85,B 0,C 180,E1 -17146.359,E2 -17146.359} C_VEL
LIN {X 0,Y 293.228,Z 426.698,A -85,B 0,C 180,E1 -17147.852,E2 -17147.852} C_VEL
LIN {X 0,Y 291.267,Z 435.169,A -85,B 0,C 180,E1 -17149.35,E2 -17149.35} C_VEL
LIN {X 0,Y 289.158,Z 444.076,A -85,B 0,C 180,E1 -17151.302,E2 -17151.302} C_VEL
LIN {X 0,Y 287.431,Z 451.014,A -85,B 0,C 180,E1 -17153.202,E2 -17153.202} C_VEL
LIN {X 0,Y 285.703,Z 457.791,A -85,B 0,C 180,E1 -17155.547,E2 -17155.547} C_VEL
LIN {X 0,Y 284.38,Z 463.041,A -85,B 0,C 180,E1 -17157.907,E2 -17157.907} C_VEL
LIN {X 0,Y 283.436,Z 466.942,A -85,B 0,C 180,E1 -17160.273,E2 -17160.273} C_VEL
LIN {X 0,Y 282.914,Z 468.826,A -85,B 0,C 180,E1 -17161.839,E2 -17161.839} C_VEL
LIN {X 0,Y 282.485,Z 470.352,A -85,B 0,C 180,E1 -17163.575,E2 -17163.575} C_VEL
LIN {X 0,Y 282.217,Z 471.146,A -85,B 0,C 180,E1 -17164.957,E2 -17164.957} C_VEL
LIN {X 0,Y 282.006,Z 471.628,A -85,B 0,C 180,E1 -17167.214,E2 -17167.214} C_VEL
LIN {X 0,Y 281.921,Z 471.077,A -85,B 0,C 180,E1 -17169.576,E2 -17169.576} C_VEL
LIN {X 0,Y 282.003,Z 470.005,A -85,B 0,C 180,E1 -17171.243,E2 -17171.243} C_VEL
LIN {X 0,Y 282.111,Z 468.738,A -85,B 0,C 180,E1 -17172.608,E2 -17172.608} C_VEL
LIN {X 0,Y 282.458,Z 465.786,A -85,B 0,C 180,E1 -17174.858,E2 -17174.858} C_VEL
LIN {X 0,Y 282.906,Z 461.74,A -85,B 0,C 180,E1 -17177.083,E2 -17177.083} C_VEL
LIN {X 0,Y 283.508,Z 456.502,A -85,B 0,C 180,E1 -17179.288,E2 -17179.288} C_VEL
LIN {X 0,Y 284.352,Z 449.867,A -85,B 0,C 180,E1 -17181.474,E2 -17181.474} C_VEL
LIN {X 0,Y 285.514,Z 441.565,A -85,B 0,C 180,E1 -17183.643,E2 -17183.643} C_VEL
LIN {X 0,Y 286.639,Z 433.096,A -85,B 0,C 180,E1 -17185.432,E2 -17185.432} C_VEL
LIN {X 0,Y 288.005,Z 423.778,A -85,B 0,C 180,E1 -17187.03,E2 -17187.03} C_VEL
LIN {X 0,Y 289.36,Z 413.329,A -85,B 0,C 180,E1 -17188.471,E2 -17188.471} C_VEL
LIN {X 0,Y 290.704,Z 400.778,A -85,B 0,C 180,E1 -17189.829,E2 -17189.829} C_VEL
LIN {X 0,Y 291.738,Z 389.222,A -85,B 0,C 180,E1 -17190.779,E2 -17190.779} C_VEL
LIN {X 0,Y 292.624,Z 375.997,A -85,B 0,C 180,E1 -17191.55,E2 -17191.55} C_VEL
LIN {X 0,Y 293.196,Z 363.324,A -85,B 0,C 180,E1 -17192.02,E2 -17192.02} C_VEL
LIN {X 0,Y 294.773,Z 294.919,A -85,B 0,C 180,E1 -17193.703,E2 -17193.703} C_VEL
LIN {X 0,Y 291.519,Z 275.821,A -85,B 0,C 180,E1 -17194.443,E2 -17194.443} C_VEL
LIN {X 0,Y 286.264,Z 260.554,A -85,B 0,C 180,E1 -17195.293,E2 -17195.293} C_VEL
LIN {X 0,Y 284.753,Z 252.165,A -85,B 0,C 180,E1 -17198.161,E2 -17198.161} C_VEL
LIN {X 0,Y 284.605,Z 251.555,A -85,B 0,C 180,E1 -17198.523,E2 -17198.523} C_VEL
LIN {X 0,Y 284.441,Z 251.551,A -85,B 0,C 180,E1 -17202.851,E2 -17202.851} C_VEL
LIN {X 0,Y 284.448,Z 251.541,A -85,B 0,C 180,E1 -17205.773,E2 -17205.773} C_VEL
LIN {X 0,Y 284.344,Z 251.565,A -85,B 0,C 180,E1 -17210.247,E2 -17210.247} C_VEL
LIN {X 0,Y 284.28,Z 251.575,A -85,B 0,C 180,E1 -17213.853,E2 -17213.853} C_VEL
LIN {X 0,Y 284.245,Z 251.577,A -85,B 0,C 180,E1 -17218.022,E2 -17218.022} C_VEL
LIN {X 0,Y 284.256,Z 251.573,A -85,B 0,C 180,E1 -17221.281,E2 -17221.281} C_VEL
LIN {X 0,Y 284.311,Z 251.567,A -85,B 0,C 180,E1 -17225.352,E2 -17225.352} C_VEL
LIN {X 0,Y 284.271,Z 251.574,A -85,B 0,C 180,E1 -17228.178,E2 -17228.178} C_VEL
LIN {X 0,Y 284.214,Z 251.577,A -85,B 0,C 180,E1 -17232.123,E2 -17232.123} C_VEL
LIN {X 0,Y 284.219,Z 251.579,A -85,B 0,C 180,E1 -17236.192,E2 -17236.192} C_VEL
LIN {X 0,Y 284.267,Z 251.563,A -85,B 0,C 180,E1 -17240.036,E2 -17240.036} C_VEL
LIN {X 0,Y 284.306,Z 251.568,A -85,B 0,C 180,E1 -17243.619,E2 -17243.619} C_VEL
LIN {X 0,Y 284.294,Z 251.567,A -85,B 0,C 180,E1 -17247.197,E2 -17247.197} C_VEL
LIN {X 0,Y 284.299,Z 251.552,A -85,B 0,C 180,E1 -17250.377,E2 -17250.377} C_VEL
LIN {X 0,Y 284.288,Z 251.571,A -85,B 0,C 180,E1 -17253.585,E2 -17253.585} C_VEL
LIN {X 0,Y 284.303,Z 251.569,A -85,B 0,C 180,E1 -17256.708,E2 -17256.708} C_VEL
LIN {X 0,Y 284.284,Z 251.565,A -85,B 0,C 180,E1 -17259.086,E2 -17259.086} C_VEL
LIN {X 0,Y 283.668,Z 251.642,A -85,B 0,C 180,E1 -17260.268,E2 -17260.268} C_VEL
LIN {X 0,Y 280.922,Z 251.984,A -85,B 0,C 180,E1 -17262.197,E2 -17262.197} C_VEL
LIN {X 0,Y 278.554,Z 252.277,A -85,B 0,C 180,E1 -17263.762,E2 -17263.762} C_VEL
LIN {X 0,Y 277.507,Z 252.405,A -85,B 0,C 180,E1 -17264.973,E2 -17264.973} C_VEL
LIN {X 0,Y 277.406,Z 252.416,A -85,B 0,C 180,E1 -17265.384,E2 -17265.384} C_VEL
LIN {X 0,Y 277.46,Z 252.425,A -85,B 0,C 180,E1 -17269.793,E2 -17269.793} C_VEL
LIN {X 0,Y 277.604,Z 252.398,A -85,B 0,C 180,E1 -17272.734,E2 -17272.734} C_VEL
LIN {X 0,Y 277.811,Z 252.37,A -85,B 0,C 180,E1 -17278.556,E2 -17278.556} C_VEL
LIN {X 0,Y 277.817,Z 252.374,A -85,B 0,C 180,E1 -17281.455,E2 -17281.455} C_VEL
LIN {X 0,Y 277.603,Z 252.395,A -85,B 0,C 180,E1 -17287.278,E2 -17287.278} C_VEL
LIN {X 0,Y 277.466,Z 252.404,A -85,B 0,C 180,E1 -17290.218,E2 -17290.218} C_VEL
LIN {X 0,Y 277.424,Z 252.43,A -85,B 0,C 180,E1 -17294.68,E2 -17294.68} C_VEL
LIN {X 0,Y 277.301,Z 252.431,A -85,B 0,C 180,E1 -17299.242,E2 -17299.242} C_VEL
LIN {X 0,Y 277.298,Z 252.44,A -85,B 0,C 180,E1 -17303.928,E2 -17303.928} C_VEL
LIN {X 0,Y 277.286,Z 252.44,A -85,B 0,C 180,E1 -17307.485,E2 -17307.485} C_VEL
LIN {X 0,Y 277.266,Z 252.437,A -85,B 0,C 180,E1 -17310.476,E2 -17310.476} C_VEL
LIN {X 0,Y 277.264,Z 252.446,A -85,B 0,C 180,E1 -17313.899,E2 -17313.899} C_VEL
LIN {X 0,Y 277.251,Z 252.444,A -85,B 0,C 180,E1 -17317.477,E2 -17317.477} C_VEL
LIN {X 0,Y 277.195,Z 252.457,A -85,B 0,C 180,E1 -17321.245,E2 -17321.245} C_VEL
LIN {X 0,Y 277.193,Z 252.457,A -85,B 0,C 180,E1 -17325.234,E2 -17325.234} C_VEL
LIN {X 0,Y 277.216,Z 252.455,A -85,B 0,C 180,E1 -17329.52,E2 -17329.52} C_VEL
LIN {X 0,Y 277.27,Z 252.443,A -85,B 0,C 180,E1 -17332.529,E2 -17332.529} C_VEL
LIN {X 0,Y 277.265,Z 252.443,A -85,B 0,C 180,E1 -17336.104,E2 -17336.104} C_VEL
LIN {X 0,Y 277.32,Z 252.569,A -85,B 0,C 180,E1 -17338.041,E2 -17338.041} C_VEL
LIN {X 0,Y 279.278,Z 261.99,A -85,B 0,C 180,E1 -17341.434,E2 -17341.434} C_VEL
LIN {X 0,Y 280.393,Z 267.659,A -85,B 0,C 180,E1 -17343.265,E2 -17343.265} C_VEL
LIN {X 0,Y 283.202,Z 276.085,A -85,B 0,C 180,E1 -17343.774,E2 -17343.774} C_VEL
LIN {X 0,Y 288.016,Z 309.462,A -85,B 0,C 180,E1 -17345.034,E2 -17345.034} C_VEL
LIN {X 0,Y 286.258,Z 375.873,A -85,B 0,C 180,E1 -17346.734,E2 -17346.734} C_VEL
LIN {X 0,Y 285.397,Z 389.512,A -85,B 0,C 180,E1 -17347.368,E2 -17347.368} C_VEL
LIN {X 0,Y 284.338,Z 402.002,A -85,B 0,C 180,E1 -17348.236,E2 -17348.236} C_VEL
LIN {X 0,Y 282.898,Z 414.737,A -85,B 0,C 180,E1 -17349.455,E2 -17349.455} C_VEL
LIN {X 0,Y 281.451,Z 426.074,A -85,B 0,C 180,E1 -17350.866,E2 -17350.866} C_VEL
LIN {X 0,Y 280.167,Z 436.278,A -85,B 0,C 180,E1 -17352.479,E2 -17352.479} C_VEL
LIN {X 0,Y 278.813,Z 445.458,A -85,B 0,C 180,E1 -17354.276,E2 -17354.276} C_VEL
LIN {X 0,Y 277.52,Z 454.399,A -85,B 0,C 180,E1 -17356.45,E2 -17356.45} C_VEL
LIN {X 0,Y 276.55,Z 461.542,A -85,B 0,C 180,E1 -17358.639,E2 -17358.639} C_VEL
LIN {X 0,Y 275.762,Z 468.039,A -85,B 0,C 180,E1 -17361.202,E2 -17361.202} C_VEL
LIN {X 0,Y 275.415,Z 472.308,A -85,B 0,C 180,E1 -17363.404,E2 -17363.404} C_VEL
LIN {X 0,Y 275.234,Z 475.487,A -85,B 0,C 180,E1 -17365.604,E2 -17365.604} C_VEL
LIN {X 0,Y 275.223,Z 477.066,A -85,B 0,C 180,E1 -17367.07,E2 -17367.07} C_VEL
LIN {X 0,Y 275.232,Z 478.215,A -85,B 0,C 180,E1 -17368.535,E2 -17368.535} C_VEL
LIN {X 0,Y 275.229,Z 478.926,A -85,B 0,C 180,E1 -17369.998,E2 -17369.998} C_VEL
LIN {X 0,Y 275.232,Z 479.25,A -85,B 0,C 180,E1 -17371.461,E2 -17371.461} C_VEL
LIN {X 0,Y 275.227,Z 479.19,A -85,B 0,C 180,E1 -17372.925,E2 -17372.925} C_VEL
LIN {X 0,Y 275.352,Z 478.153,A -85,B 0,C 180,E1 -17375.449,E2 -17375.449} C_VEL
LIN {X 0,Y 275.62,Z 476.587,A -85,B 0,C 180,E1 -17377.322,E2 -17377.322} C_VEL
LIN {X 0,Y 276.208,Z 473.912,A -85,B 0,C 180,E1 -17379.518,E2 -17379.518} C_VEL
LIN {X 0,Y 277.057,Z 470.242,A -85,B 0,C 180,E1 -17381.706,E2 -17381.706} C_VEL
LIN {X 0,Y 278.287,Z 465.482,A -85,B 0,C 180,E1 -17383.879,E2 -17383.879} C_VEL
LIN {X 0,Y 279.974,Z 459.488,A -85,B 0,C 180,E1 -17386.027,E2 -17386.027} C_VEL
LIN {X 0,Y 282.006,Z 452.049,A -85,B 0,C 180,E1 -17388.148,E2 -17388.148} C_VEL
LIN {X 0,Y 283.738,Z 444.752,A -85,B 0,C 180,E1 -17389.849,E2 -17389.849} C_VEL
LIN {X 0,Y 285.992,Z 435.352,A -85,B 0,C 180,E1 -17391.627,E2 -17391.627} C_VEL
LIN {X 0,Y 288.165,Z 425.215,A -85,B 0,C 180,E1 -17393.156,E2 -17393.156} C_VEL
LIN {X 0,Y 290.36,Z 414.003,A -85,B 0,C 180,E1 -17394.485,E2 -17394.485} C_VEL
LIN {X 0,Y 292.059,Z 403.402,A -85,B 0,C 180,E1 -17395.474,E2 -17395.474} C_VEL
LIN {X 0,Y 293.761,Z 390.601,A -85,B 0,C 180,E1 -17396.363,E2 -17396.363} C_VEL
LIN {X 0,Y 294.997,Z 377.558,A -85,B 0,C 180,E1 -17396.968,E2 -17396.968} C_VEL
LIN {X 0,Y 295.917,Z 356.324,A -85,B 0,C 180,E1 -17397.552,E2 -17397.552} C_VEL
LIN {X 0,Y 297.421,Z 311.581,A -85,B 0,C 180,E1 -17398.68,E2 -17398.68} C_VEL
LIN {X 0,Y 294.137,Z 293.874,A -85,B 0,C 180,E1 -17399.654,E2 -17399.654} C_VEL
LIN {X 0,Y 287.41,Z 279.167,A -85,B 0,C 180,E1 -17401.072,E2 -17401.072} C_VEL
LIN {X 0,Y 281.045,Z 266.94,A -85,B 0,C 180,E1 -17402.496,E2 -17402.496} C_VEL
LIN {X 0,Y 279.756,Z 261.719,A -85,B 0,C 180,E1 -17404.539,E2 -17404.539} C_VEL
LIN {X 0,Y 278.039,Z 255.346,A -85,B 0,C 180,E1 -17407.344,E2 -17407.344} C_VEL
LIN {X 0,Y 277.262,Z 252.48,A -85,B 0,C 180,E1 -17408.775,E2 -17408.775} C_VEL
LIN {X 0,Y 277.21,Z 252.443,A -85,B 0,C 180,E1 -17413.194,E2 -17413.194} C_VEL
LIN {X 0,Y 277.195,Z 252.435,A -85,B 0,C 180,E1 -17417.326,E2 -17417.326} C_VEL
LIN {X 0,Y 277.251,Z 252.448,A -85,B 0,C 180,E1 -17421.792,E2 -17421.792} C_VEL
LIN {X 0,Y 277.278,Z 252.44,A -85,B 0,C 180,E1 -17424.335,E2 -17424.335} C_VEL
LIN {X 0,Y 277.239,Z 252.445,A -85,B 0,C 180,E1 -17427.831,E2 -17427.831} C_VEL
LIN {X 0,Y 277.237,Z 252.443,A -85,B 0,C 180,E1 -17431.201,E2 -17431.201} C_VEL
LIN {X 0,Y 277.233,Z 252.443,A -85,B 0,C 180,E1 -17434.466,E2 -17434.466} C_VEL
LIN {X 0,Y 277.245,Z 252.447,A -85,B 0,C 180,E1 -17437.646,E2 -17437.646} C_VEL
LIN {X 0,Y 277.279,Z 252.445,A -85,B 0,C 180,E1 -17440.756,E2 -17440.756} C_VEL
LIN {X 0,Y 277.402,Z 252.432,A -85,B 0,C 180,E1 -17445.319,E2 -17445.319} C_VEL
LIN {X 0,Y 277.448,Z 252.425,A -85,B 0,C 180,E1 -17449.781,E2 -17449.781} C_VEL
LIN {X 0,Y 277.594,Z 252.393,A -85,B 0,C 180,E1 -17452.722,E2 -17452.722} C_VEL
LIN {X 0,Y 277.796,Z 252.38,A -85,B 0,C 180,E1 -17458.545,E2 -17458.545} C_VEL
LIN {X 0,Y 277.79,Z 252.371,A -85,B 0,C 180,E1 -17461.444,E2 -17461.444} C_VEL
LIN {X 0,Y 277.582,Z 252.407,A -85,B 0,C 180,E1 -17467.267,E2 -17467.267} C_VEL
LIN {X 0,Y 277.439,Z 252.419,A -85,B 0,C 180,E1 -17470.208,E2 -17470.208} C_VEL
LIN {X 0,Y 277.389,Z 252.433,A -85,B 0,C 180,E1 -17474.67,E2 -17474.67} C_VEL
LIN {X 0,Y 277.301,Z 252.44,A -85,B 0,C 180,E1 -17479.23,E2 -17479.23} C_VEL
LIN {X 0,Y 277.273,Z 252.448,A -85,B 0,C 180,E1 -17483.918,E2 -17483.918} C_VEL
LIN {X 0,Y 277.298,Z 252.433,A -85,B 0,C 180,E1 -17487.5,E2 -17487.5} C_VEL
LIN {X 0,Y 277.244,Z 252.449,A -85,B 0,C 180,E1 -17490.477,E2 -17490.477} C_VEL
LIN {X 0,Y 277.224,Z 252.566,A -85,B 0,C 180,E1 -17492.618,E2 -17492.618} C_VEL
LIN {X 0,Y 279.317,Z 259.997,A -85,B 0,C 180,E1 -17496.021,E2 -17496.021} C_VEL
LIN {X 0,Y 279.73,Z 261.246,A -85,B 0,C 180,E1 -17496.363,E2 -17496.363} C_VEL
LIN {X 0,Y 286.95,Z 274.405,A -85,B 0,C 180,E1 -17497.946,E2 -17497.946} C_VEL
LIN {X 0,Y 293.082,Z 286.891,A -85,B 0,C 180,E1 -17499.223,E2 -17499.223} C_VEL
LIN {X 0,Y 296.975,Z 296.135,A -85,B 0,C 180,E1 -17500.037,E2 -17500.037} C_VEL
LIN {X 0,Y 297.828,Z 300.665,A -85,B 0,C 180,E1 -17500.286,E2 -17500.286} C_VEL
LIN {X 0,Y 295.237,Z 368.919,A -85,B 0,C 180,E1 -17502.019,E2 -17502.019} C_VEL
LIN {X 0,Y 294.102,Z 382.674,A -85,B 0,C 180,E1 -17502.649,E2 -17502.649} C_VEL
LIN {X 0,Y 292.738,Z 394.312,A -85,B 0,C 180,E1 -17503.432,E2 -17503.432} C_VEL
LIN {X 0,Y 291.024,Z 405.564,A -85,B 0,C 180,E1 -17504.444,E2 -17504.444} C_VEL
LIN {X 0,Y 288.794,Z 417.529,A -85,B 0,C 180,E1 -17505.848,E2 -17505.848} C_VEL
LIN {X 0,Y 286.456,Z 428.42,A -85,B 0,C 180,E1 -17507.484,E2 -17507.484} C_VEL
LIN {X 0,Y 284.379,Z 436.969,A -85,B 0,C 180,E1 -17509.091,E2 -17509.091} C_VEL
LIN {X 0,Y 282.197,Z 445.572,A -85,B 0,C 180,E1 -17511.106,E2 -17511.106} C_VEL
LIN {X 0,Y 280.186,Z 453.254,A -85,B 0,C 180,E1 -17513.373,E2 -17513.373} C_VEL
LIN {X 0,Y 278.66,Z 458.767,A -85,B 0,C 180,E1 -17515.429,E2 -17515.429} C_VEL
LIN {X 0,Y 277.298,Z 463.808,A -85,B 0,C 180,E1 -17517.846,E2 -17517.846} C_VEL
LIN {X 0,Y 276.51,Z 466.837,A -85,B 0,C 180,E1 -17519.773,E2 -17519.773} C_VEL
LIN {X 0,Y 276.04,Z 468.465,A -85,B 0,C 180,E1 -17521.073,E2 -17521.073} C_VEL
LIN {X 0,Y 275.475,Z 470.395,A -85,B 0,C 180,E1 -17523.227,E2 -17523.227} C_VEL
LIN {X 0,Y 274.993,Z 471.609,A -85,B 0,C 180,E1 -17525.866,E2 -17525.866} C_VEL
LIN {X 0,Y 274.899,Z 471.688,A -85,B 0,C 180,E1 -17527.453,E2 -17527.453} C_VEL
LIN {X 0,Y 274.81,Z 471.335,A -85,B 0,C 180,E1 -17529.023,E2 -17529.023} C_VEL
LIN {X 0,Y 274.883,Z 470.191,A -85,B 0,C 180,E1 -17531.059,E2 -17531.059} C_VEL
LIN {X 0,Y 275.173,Z 467.546,A -85,B 0,C 180,E1 -17533.686,E2 -17533.686} C_VEL
LIN {X 0,Y 275.528,Z 464.506,A -85,B 0,C 180,E1 -17535.729,E2 -17535.729} C_VEL
LIN {X 0,Y 276.084,Z 459.471,A -85,B 0,C 180,E1 -17538.252,E2 -17538.252} C_VEL
LIN {X 0,Y 276.8,Z 453.602,A -85,B 0,C 180,E1 -17540.503,E2 -17540.503} C_VEL
LIN {X 0,Y 277.8,Z 446.2,A -85,B 0,C 180,E1 -17542.735,E2 -17542.735} C_VEL
LIN {X 0,Y 279.231,Z 436.95,A -85,B 0,C 180,E1 -17544.948,E2 -17544.948} C_VEL
LIN {X 0,Y 280.571,Z 427.396,A -85,B 0,C 180,E1 -17546.771,E2 -17546.771} C_VEL
LIN {X 0,Y 282.039,Z 417.067,A -85,B 0,C 180,E1 -17548.344,E2 -17548.344} C_VEL
LIN {X 0,Y 283.27,Z 406.429,A -85,B 0,C 180,E1 -17549.647,E2 -17549.647} C_VEL
LIN {X 0,Y 284.479,Z 394.37,A -85,B 0,C 180,E1 -17550.798,E2 -17550.798} C_VEL
LIN {X 0,Y 285.545,Z 381.65,A -85,B 0,C 180,E1 -17551.677,E2 -17551.677} C_VEL
LIN {X 0,Y 286.232,Z 368.674,A -85,B 0,C 180,E1 -17552.289,E2 -17552.289} C_VEL
LIN {X 0,Y 287.999,Z 304.421,A -85,B 0,C 180,E1 -17553.941,E2 -17553.941} C_VEL
LIN {X 0,Y 288.126,Z 295.805,A -85,B 0,C 180,E1 -17554.163,E2 -17554.163} C_VEL
LIN {X 0,Y 285.083,Z 277.858,A -85,B 0,C 180,E1 -17554.879,E2 -17554.879} C_VEL
LIN {X 0,Y 279.1,Z 260.539,A -85,B 0,C 180,E1 -17555.874,E2 -17555.874} C_VEL
LIN {X 0,Y 278.031,Z 254.48,A -85,B 0,C 180,E1 -17557.994,E2 -17557.994} C_VEL
LIN {X 0,Y 277.573,Z 252.432,A -85,B 0,C 180,E1 -17558.873,E2 -17558.873} C_VEL
LIN {X 0,Y 277.381,Z 252.432,A -85,B 0,C 180,E1 -17563.183,E2 -17563.183} C_VEL
LIN {X 0,Y 277.367,Z 252.419,A -85,B 0,C 180,E1 -17566.186,E2 -17566.186} C_VEL
LIN {X 0,Y 277.288,Z 252.443,A -85,B 0,C 180,E1 -17570.34,E2 -17570.34} C_VEL
LIN {X 0,Y 277.222,Z 252.455,A -85,B 0,C 180,E1 -17574.144,E2 -17574.144} C_VEL
LIN {X 0,Y 277.213,Z 252.45,A -85,B 0,C 180,E1 -17577.477,E2 -17577.477} C_VEL
LIN {X 0,Y 277.221,Z 252.452,A -85,B 0,C 180,E1 -17580.478,E2 -17580.478} C_VEL
LIN {X 0,Y 277.22,Z 252.448,A -85,B 0,C 180,E1 -17583.902,E2 -17583.902} C_VEL
LIN {X 0,Y 277.226,Z 252.449,A -85,B 0,C 180,E1 -17587.478,E2 -17587.478} C_VEL
LIN {X 0,Y 277.161,Z 252.454,A -85,B 0,C 180,E1 -17591.248,E2 -17591.248} C_VEL
LIN {X 0,Y 277.154,Z 252.459,A -85,B 0,C 180,E1 -17595.239,E2 -17595.239} C_VEL
LIN {X 0,Y 277.167,Z 252.447,A -85,B 0,C 180,E1 -17598.765,E2 -17598.765} C_VEL
LIN {X 0,Y 277.24,Z 252.447,A -85,B 0,C 180,E1 -17602.535,E2 -17602.535} C_VEL
LIN {X 0,Y 277.234,Z 252.447,A -85,B 0,C 180,E1 -17606.111,E2 -17606.111} C_VEL
LIN {X 0,Y 277.218,Z 252.435,A -85,B 0,C 180,E1 -17609.541,E2 -17609.541} C_VEL
LIN {X 0,Y 277.242,Z 252.441,A -85,B 0,C 180,E1 -17612.859,E2 -17612.859} C_VEL
LIN {X 0,Y 277.252,Z 252.447,A -85,B 0,C 180,E1 -17616.08,E2 -17616.08} C_VEL
LIN {X 0,Y 277.282,Z 252.435,A -85,B 0,C 180,E1 -17620.768,E2 -17620.768} C_VEL
LIN {X 0,Y 277.406,Z 252.416,A -85,B 0,C 180,E1 -17625.384,E2 -17625.384} C_VEL
LIN {X 0,Y 276.709,Z 252.51,A -85,B 0,C 180,E1 -17626.596,E2 -17626.596} C_VEL
LIN {X 0,Y 273.906,Z 252.863,A -85,B 0,C 180,E1 -17628.574,E2 -17628.574} C_VEL
LIN {X 0,Y 271.571,Z 253.156,A -85,B 0,C 180,E1 -17630.18,E2 -17630.18} C_VEL
LIN {X 0,Y 270.595,Z 253.277,A -85,B 0,C 180,E1 -17631.424,E2 -17631.424} C_VEL
LIN {X 0,Y 270.527,Z 253.279,A -85,B 0,C 180,E1 -17631.844,E2 -17631.844} C_VEL
LIN {X 0,Y 270.513,Z 253.277,A -85,B 0,C 180,E1 -17634.041,E2 -17634.041} C_VEL
LIN {X 0,Y 270.777,Z 253.243,A -85,B 0,C 180,E1 -17638.519,E2 -17638.519} C_VEL
LIN {X 0,Y 270.781,Z 253.251,A -85,B 0,C 180,E1 -17641.493,E2 -17641.493} C_VEL
LIN {X 0,Y 270.564,Z 253.271,A -85,B 0,C 180,E1 -17647.468,E2 -17647.468} C_VEL
LIN {X 0,Y 270.4,Z 253.285,A -85,B 0,C 180,E1 -17650.488,E2 -17650.488} C_VEL
LIN {X 0,Y 270.383,Z 253.304,A -85,B 0,C 180,E1 -17655.071,E2 -17655.071} C_VEL
LIN {X 0,Y 270.24,Z 253.308,A -85,B 0,C 180,E1 -17659.766,E2 -17659.766} C_VEL
LIN {X 0,Y 270.241,Z 253.321,A -85,B 0,C 180,E1 -17664.594,E2 -17664.594} C_VEL
LIN {X 0,Y 270.215,Z 253.318,A -85,B 0,C 180,E1 -17667.92,E2 -17667.92} C_VEL
LIN {X 0,Y 270.192,Z 253.325,A -85,B 0,C 180,E1 -17671.353,E2 -17671.353} C_VEL
LIN {X 0,Y 270.216,Z 253.325,A -85,B 0,C 180,E1 -17674.909,E2 -17674.909} C_VEL
LIN {X 0,Y 270.187,Z 253.326,A -85,B 0,C 180,E1 -17678.705,E2 -17678.705} C_VEL
LIN {X 0,Y 270.166,Z 253.325,A -85,B 0,C 180,E1 -17683.246,E2 -17683.246} C_VEL
LIN {X 0,Y 270.169,Z 253.327,A -85,B 0,C 180,E1 -17687.439,E2 -17687.439} C_VEL
LIN {X 0,Y 270.212,Z 253.319,A -85,B 0,C 180,E1 -17691.372,E2 -17691.372} C_VEL
LIN {X 0,Y 270.217,Z 253.321,A -85,B 0,C 180,E1 -17695.094,E2 -17695.094} C_VEL
LIN {X 0,Y 270.266,Z 253.492,A -85,B 0,C 180,E1 -17697.673,E2 -17697.673} C_VEL
LIN {X 0,Y 272.34,Z 263.472,A -85,B 0,C 180,E1 -17701.339,E2 -17701.339} C_VEL
LIN {X 0,Y 273.175,Z 267.573,A -85,B 0,C 180,E1 -17702.674,E2 -17702.674} C_VEL
LIN {X 0,Y 276.846,Z 278.8,A -85,B 0,C 180,E1 -17703.349,E2 -17703.349} C_VEL
LIN {X 0,Y 281.33,Z 310.26,A -85,B 0,C 180,E1 -17704.568,E2 -17704.568} C_VEL
LIN {X 0,Y 279.516,Z 375.636,A -85,B 0,C 180,E1 -17706.276,E2 -17706.276} C_VEL
LIN {X 0,Y 278.631,Z 389.478,A -85,B 0,C 180,E1 -17706.934,E2 -17706.934} C_VEL
LIN {X 0,Y 277.495,Z 402.461,A -85,B 0,C 180,E1 -17707.866,E2 -17707.866} C_VEL
LIN {X 0,Y 276.003,Z 415.07,A -85,B 0,C 180,E1 -17709.113,E2 -17709.113} C_VEL
LIN {X 0,Y 274.518,Z 426.328,A -85,B 0,C 180,E1 -17710.558,E2 -17710.558} C_VEL
LIN {X 0,Y 273.316,Z 435.728,A -85,B 0,C 180,E1 -17712.078,E2 -17712.078} C_VEL
LIN {X 0,Y 271.964,Z 444.763,A -85,B 0,C 180,E1 -17713.869,E2 -17713.869} C_VEL
LIN {X 0,Y 270.585,Z 453.803,A -85,B 0,C 180,E1 -17716.096,E2 -17716.096} C_VEL
LIN {X 0,Y 269.549,Z 461.062,A -85,B 0,C 180,E1 -17718.34,E2 -17718.34} C_VEL
LIN {X 0,Y 268.945,Z 465.949,A -85,B 0,C 180,E1 -17720.218,E2 -17720.218} C_VEL
LIN {X 0,Y 268.442,Z 470.678,A -85,B 0,C 180,E1 -17722.476,E2 -17722.476} C_VEL
LIN {X 0,Y 268.202,Z 474.304,A -85,B 0,C 180,E1 -17724.759,E2 -17724.759} C_VEL
LIN {X 0,Y 268.138,Z 476.836,A -85,B 0,C 180,E1 -17726.993,E2 -17726.993} C_VEL
LIN {X 0,Y 268.138,Z 478.033,A -85,B 0,C 180,E1 -17728.496,E2 -17728.496} C_VEL
LIN {X 0,Y 268.155,Z 478.784,A -85,B 0,C 180,E1 -17729.998,E2 -17729.998} C_VEL
LIN {X 0,Y 268.138,Z 479.137,A -85,B 0,C 180,E1 -17731.5,E2 -17731.5} C_VEL
LIN {X 0,Y 268.124,Z 479.105,A -85,B 0,C 180,E1 -17733.003,E2 -17733.003} C_VEL
LIN {X 0,Y 268.233,Z 478.278,A -85,B 0,C 180,E1 -17735.312,E2 -17735.312} C_VEL
LIN {X 0,Y 268.56,Z 476.618,A -85,B 0,C 180,E1 -17737.516,E2 -17737.516} C_VEL
LIN {X 0,Y 269.458,Z 472.934,A -85,B 0,C 180,E1 -17740.517,E2 -17740.517} C_VEL
LIN {X 0,Y 270.53,Z 468.973,A -85,B 0,C 180,E1 -17742.755,E2 -17742.755} C_VEL
LIN {X 0,Y 271.89,Z 463.9,A -85,B 0,C 180,E1 -17744.978,E2 -17744.978} C_VEL
LIN {X 0,Y 273.831,Z 457.529,A -85,B 0,C 180,E1 -17747.164,E2 -17747.164} C_VEL
LIN {X 0,Y 275.914,Z 449.613,A -85,B 0,C 180,E1 -17749.335,E2 -17749.335} C_VEL
LIN {X 0,Y 277.965,Z 441.571,A -85,B 0,C 180,E1 -17751.116,E2 -17751.116} C_VEL
LIN {X 0,Y 280.411,Z 431.797,A -85,B 0,C 180,E1 -17752.857,E2 -17752.857} C_VEL
LIN {X 0,Y 282.804,Z 420.89,A -85,B 0,C 180,E1 -17754.4,E2 -17754.4} C_VEL
LIN {X 0,Y 284.904,Z 410.234,A -85,B 0,C 180,E1 -17755.572,E2 -17755.572} C_VEL
LIN {X 0,Y 286.679,Z 398.595,A -85,B 0,C 180,E1 -17756.574,E2 -17756.574} C_VEL
LIN {X 0,Y 288.302,Z 385.376,A -85,B 0,C 180,E1 -17757.392,E2 -17757.392} C_VEL
LIN {X 0,Y 289.389,Z 372.456,A -85,B 0,C 180,E1 -17757.893,E2 -17757.893} C_VEL
LIN {X 0,Y 291.541,Z 312.731,A -85,B 0,C 180,E1 -17759.437,E2 -17759.437} C_VEL
LIN {X 0,Y 288.683,Z 296.931,A -85,B 0,C 180,E1 -17760.328,E2 -17760.328} C_VEL
LIN {X 0,Y 282.428,Z 283.146,A -85,B 0,C 180,E1 -17761.701,E2 -17761.701} C_VEL
LIN {X 0,Y 275.556,Z 270.271,A -85,B 0,C 180,E1 -17763.247,E2 -17763.247} C_VEL
LIN {X 0,Y 273.751,Z 266.545,A -85,B 0,C 180,E1 -17763.776,E2 -17763.776} C_VEL
LIN {X 0,Y 272.021,Z 259.572,A -85,B 0,C 180,E1 -17766.775,E2 -17766.775} C_VEL
LIN {X 0,Y 270.194,Z 253.367,A -85,B 0,C 180,E1 -17769.857,E2 -17769.857} C_VEL
LIN {X 0,Y 270.166,Z 253.321,A -85,B 0,C 180,E1 -17773.243,E2 -17773.243} C_VEL
LIN {X 0,Y 270.154,Z 253.312,A -85,B 0,C 180,E1 -17777.432,E2 -17777.432} C_VEL
LIN {X 0,Y 270.194,Z 253.324,A -85,B 0,C 180,E1 -17781.366,E2 -17781.366} C_VEL
LIN {X 0,Y 270.198,Z 253.328,A -85,B 0,C 180,E1 -17785.089,E2 -17785.089} C_VEL
LIN {X 0,Y 270.184,Z 253.33,A -85,B 0,C 180,E1 -17789.131,E2 -17789.131} C_VEL
LIN {X 0,Y 270.22,Z 253.323,A -85,B 0,C 180,E1 -17792.158,E2 -17792.158} C_VEL
LIN {X 0,Y 270.181,Z 253.323,A -85,B 0,C 180,E1 -17795.558,E2 -17795.558} C_VEL
LIN {X 0,Y 270.218,Z 253.321,A -85,B 0,C 180,E1 -17800.233,E2 -17800.233} C_VEL
LIN {X 0,Y 270.362,Z 253.305,A -85,B 0,C 180,E1 -17804.928,E2 -17804.928} C_VEL
LIN {X 0,Y 270.401,Z 253.301,A -85,B 0,C 180,E1 -17809.512,E2 -17809.512} C_VEL
LIN {X 0,Y 270.555,Z 253.269,A -85,B 0,C 180,E1 -17812.532,E2 -17812.532} C_VEL
LIN {X 0,Y 270.76,Z 253.256,A -85,B 0,C 180,E1 -17818.507,E2 -17818.507} C_VEL
LIN {X 0,Y 270.755,Z 253.247,A -85,B 0,C 180,E1 -17821.482,E2 -17821.482} C_VEL
LIN {X 0,Y 270.544,Z 253.285,A -85,B 0,C 180,E1 -17827.457,E2 -17827.457} C_VEL
LIN {X 0,Y 270.391,Z 253.299,A -85,B 0,C 180,E1 -17830.477,E2 -17830.477} C_VEL
LIN {X 0,Y 270.357,Z 253.309,A -85,B 0,C 180,E1 -17835.061,E2 -17835.061} C_VEL
LIN {X 0,Y 270.238,Z 253.317,A -85,B 0,C 180,E1 -17839.753,E2 -17839.753} C_VEL
LIN {X 0,Y 270.213,Z 253.324,A -85,B 0,C 180,E1 -17844.584,E2 -17844.584} C_VEL
LIN {X 0,Y 270.244,Z 253.307,A -85,B 0,C 180,E1 -17847.904,E2 -17847.904} C_VEL
LIN {X 0,Y 270.168,Z 253.47,A -85,B 0,C 180,E1 -17851.561,E2 -17851.561} C_VEL
LIN {X 0,Y 272.262,Z 260.761,A -85,B 0,C 180,E1 -17854.989,E2 -17854.989} C_VEL
LIN {X 0,Y 274.492,Z 264.819,A -85,B 0,C 180,E1 -17855.617,E2 -17855.617} C_VEL
LIN {X 0,Y 281.845,Z 278.108,A -85,B 0,C 180,E1 -17857.282,E2 -17857.282} C_VEL
LIN {X 0,Y 288.12,Z 291.12,A -85,B 0,C 180,E1 -17858.645,E2 -17858.645} C_VEL
LIN {X 0,Y 291.49,Z 299.382,A -85,B 0,C 180,E1 -17859.383,E2 -17859.383} C_VEL
LIN {X 0,Y 292.001,Z 302.149,A -85,B 0,C 180,E1 -17859.539,E2 -17859.539} C_VEL
LIN {X 0,Y 289.32,Z 368.703,A -85,B 0,C 180,E1 -17861.249,E2 -17861.249} C_VEL
LIN {X 0,Y 288.174,Z 382.361,A -85,B 0,C 180,E1 -17861.879,E2 -17861.879} C_VEL
LIN {X 0,Y 286.725,Z 394.047,A -85,B 0,C 180,E1 -17862.668,E2 -17862.668} C_VEL
LIN {X 0,Y 284.99,Z 405.045,A -85,B 0,C 180,E1 -17863.659,E2 -17863.659} C_VEL
LIN {X 0,Y 282.916,Z 415.952,A -85,B 0,C 180,E1 -17864.933,E2 -17864.933} C_VEL
LIN {X 0,Y 280.438,Z 427.178,A -85,B 0,C 180,E1 -17866.605,E2 -17866.605} C_VEL
LIN {X 0,Y 277.967,Z 436.859,A -85,B 0,C 180,E1 -17868.421,E2 -17868.421} C_VEL
LIN {X 0,Y 275.714,Z 445.272,A -85,B 0,C 180,E1 -17870.416,E2 -17870.416} C_VEL
LIN {X 0,Y 273.523,Z 453.193,A -85,B 0,C 180,E1 -17872.787,E2 -17872.787} C_VEL
LIN {X 0,Y 271.62,Z 459.695,A -85,B 0,C 180,E1 -17875.306,E2 -17875.306} C_VEL
LIN {X 0,Y 270.231,Z 464.509,A -85,B 0,C 180,E1 -17877.784,E2 -17877.784} C_VEL
LIN {X 0,Y 269.212,Z 468.023,A -85,B 0,C 180,E1 -17880.267,E2 -17880.267} C_VEL
LIN {X 0,Y 268.439,Z 470.451,A -85,B 0,C 180,E1 -17882.875,E2 -17882.875} C_VEL
LIN {X 0,Y 267.987,Z 471.575,A -85,B 0,C 180,E1 -17885.193,E2 -17885.193} C_VEL
LIN {X 0,Y 267.84,Z 471.828,A -85,B 0,C 180,E1 -17886.825,E2 -17886.825} C_VEL
LIN {X 0,Y 267.72,Z 471.58,A -85,B 0,C 180,E1 -17888.44,E2 -17888.44} C_VEL
LIN {X 0,Y 267.778,Z 470.381,A -85,B 0,C 180,E1 -17890.857,E2 -17890.857} C_VEL
LIN {X 0,Y 268.122,Z 467.217,A -85,B 0,C 180,E1 -17894.027,E2 -17894.027} C_VEL
LIN {X 0,Y 268.566,Z 463.577,A -85,B 0,C 180,E1 -17896.38,E2 -17896.38} C_VEL
LIN {X 0,Y 269.126,Z 458.774,A -85,B 0,C 180,E1 -17898.708,E2 -17898.708} C_VEL
LIN {X 0,Y 269.921,Z 452.663,A -85,B 0,C 180,E1 -17901.015,E2 -17901.015} C_VEL
LIN {X 0,Y 271.009,Z 445.033,A -85,B 0,C 180,E1 -17903.301,E2 -17903.301} C_VEL
LIN {X 0,Y 272.241,Z 437.214,A -85,B 0,C 180,E1 -17905.19,E2 -17905.19} C_VEL
LIN {X 0,Y 273.632,Z 427.707,A -85,B 0,C 180,E1 -17907.058,E2 -17907.058} C_VEL
LIN {X 0,Y 275.185,Z 417.04,A -85,B 0,C 180,E1 -17908.722,E2 -17908.722} C_VEL
LIN {X 0,Y 276.627,Z 405.214,A -85,B 0,C 180,E1 -17910.184,E2 -17910.184} C_VEL
LIN {X 0,Y 277.774,Z 393.772,A -85,B 0,C 180,E1 -17911.271,E2 -17911.271} C_VEL
LIN {X 0,Y 278.87,Z 380.8,A -85,B 0,C 180,E1 -17912.169,E2 -17912.169} C_VEL
LIN {X 0,Y 279.57,Z 367.36,A -85,B 0,C 180,E1 -17912.794,E2 -17912.794} C_VEL
LIN {X 0,Y 281.406,Z 296.536,A -85,B 0,C 180,E1 -17914.645,E2 -17914.645} C_VEL
LIN {X 0,Y 278.59,Z 279.702,A -85,B 0,C 180,E1 -17915.334,E2 -17915.334} C_VEL
LIN {X 0,Y 272.005,Z 260.759,A -85,B 0,C 180,E1 -17916.447,E2 -17916.447} C_VEL
LIN {X 0,Y 270.59,Z 253.793,A -85,B 0,C 180,E1 -17918.968,E2 -17918.968} C_VEL
LIN {X 0,Y 270.468,Z 253.291,A -85,B 0,C 180,E1 -17919.463,E2 -17919.463} C_VEL
LIN {X 0,Y 270.323,Z 253.314,A -85,B 0,C 180,E1 -17923.534,E2 -17923.534} C_VEL
LIN {X 0,Y 270.299,Z 253.298,A -85,B 0,C 180,E1 -17926.621,E2 -17926.621} C_VEL
LIN {X 0,Y 270.245,Z 253.32,A -85,B 0,C 180,E1 -17930.597,E2 -17930.597} C_VEL
LIN {X 0,Y 270.154,Z 253.333,A -85,B 0,C 180,E1 -17934.599,E2 -17934.599} C_VEL
LIN {X 0,Y 270.16,Z 253.331,A -85,B 0,C 180,E1 -17937.923,E2 -17937.923} C_VEL
LIN {X 0,Y 270.147,Z 253.331,A -85,B 0,C 180,E1 -17941.355,E2 -17941.355} C_VEL
LIN {X 0,Y 270.172,Z 253.33,A -85,B 0,C 180,E1 -17944.912,E2 -17944.912} C_VEL
LIN {X 0,Y 270.176,Z 253.322,A -85,B 0,C 180,E1 -17948.717,E2 -17948.717} C_VEL
LIN {X 0,Y 270.127,Z 253.335,A -85,B 0,C 180,E1 -17953.251,E2 -17953.251} C_VEL
LIN {X 0,Y 270.133,Z 253.325,A -85,B 0,C 180,E1 -17957.444,E2 -17957.444} C_VEL
LIN {X 0,Y 270.193,Z 253.324,A -85,B 0,C 180,E1 -17961.381,E2 -17961.381} C_VEL
LIN {X 0,Y 270.185,Z 253.33,A -85,B 0,C 180,E1 -17965.101,E2 -17965.101} C_VEL
LIN {X 0,Y 270.161,Z 253.315,A -85,B 0,C 180,E1 -17969.148,E2 -17969.148} C_VEL
LIN {X 0,Y 270.179,Z 253.318,A -85,B 0,C 180,E1 -17972.184,E2 -17972.184} C_VEL
LIN {X 0,Y 270.177,Z 253.331,A -85,B 0,C 180,E1 -17975.571,E2 -17975.571} C_VEL
LIN {X 0,Y 270.22,Z 253.314,A -85,B 0,C 180,E1 -17980.245,E2 -17980.245} C_VEL
LIN {X 0,Y 270.368,Z 253.29,A -85,B 0,C 180,E1 -17984.94,E2 -17984.94} C_VEL
LIN {X 0,Y 270.412,Z 253.3,A -85,B 0,C 180,E1 -17989.524,E2 -17989.524} C_VEL
LIN {X 0,Y 270.527,Z 253.279,A -85,B 0,C 180,E1 -17991.844,E2 -17991.844} C_VEL
LIN {X 0,Y 269.87,Z 253.363,A -85,B 0,C 180,E1 -17993.085,E2 -17993.085} C_VEL
LIN {X 0,Y 266.989,Z 253.711,A -85,B 0,C 180,E1 -17995.107,E2 -17995.107} C_VEL
LIN {X 0,Y 264.624,Z 253.998,A -85,B 0,C 180,E1 -17996.751,E2 -17996.751} C_VEL
LIN {X 0,Y 263.738,Z 254.112,A -85,B 0,C 180,E1 -17998.026,E2 -17998.026} C_VEL
LIN {X 0,Y 263.736,Z 254.118,A -85,B 0,C 180,E1 -17998.457,E2 -17998.457} C_VEL
LIN {X 0,Y 263.744,Z 254.127,A -85,B 0,C 180,E1 -18001.533,E2 -18001.533} C_VEL
LIN {X 0,Y 263.525,Z 254.147,A -85,B 0,C 180,E1 -18007.669,E2 -18007.669} C_VEL
LIN {X 0,Y 263.346,Z 254.165,A -85,B 0,C 180,E1 -18010.772,E2 -18010.772} C_VEL
LIN {X 0,Y 263.325,Z 254.182,A -85,B 0,C 180,E1 -18015.485,E2 -18015.485} C_VEL
LIN {X 0,Y 263.225,Z 254.181,A -85,B 0,C 180,E1 -18020.315,E2 -18020.315} C_VEL
LIN {X 0,Y 263.184,Z 254.202,A -85,B 0,C 180,E1 -18025.299,E2 -18025.299} C_VEL
LIN {X 0,Y 263.148,Z 254.198,A -85,B 0,C 180,E1 -18028.739,E2 -18028.739} C_VEL
LIN {X 0,Y 263.147,Z 254.203,A -85,B 0,C 180,E1 -18032.292,E2 -18032.292} C_VEL
LIN {X 0,Y 263.172,Z 254.194,A -85,B 0,C 180,E1 -18035.986,E2 -18035.986} C_VEL
LIN {X 0,Y 263.091,Z 254.213,A -85,B 0,C 180,E1 -18039.881,E2 -18039.881} C_VEL
LIN {X 0,Y 263.096,Z 254.213,A -85,B 0,C 180,E1 -18043.996,E2 -18043.996} C_VEL
LIN {X 0,Y 263.099,Z 254.211,A -85,B 0,C 180,E1 -18048.419,E2 -18048.419} C_VEL
LIN {X 0,Y 263.15,Z 254.198,A -85,B 0,C 180,E1 -18052.099,E2 -18052.099} C_VEL
LIN {X 0,Y 263.172,Z 254.197,A -85,B 0,C 180,E1 -18055.886,E2 -18055.886} C_VEL
LIN {X 0,Y 263.231,Z 254.396,A -85,B 0,C 180,E1 -18057.269,E2 -18057.269} C_VEL
LIN {X 0,Y 265.286,Z 264.191,A -85,B 0,C 180,E1 -18060.963,E2 -18060.963} C_VEL
LIN {X 0,Y 265.956,Z 267.527,A -85,B 0,C 180,E1 -18062.052,E2 -18062.052} C_VEL
LIN {X 0,Y 270.451,Z 281.035,A -85,B 0,C 180,E1 -18062.885,E2 -18062.885} C_VEL
LIN {X 0,Y 274.671,Z 310.747,A -85,B 0,C 180,E1 -18064.074,E2 -18064.074} C_VEL
LIN {X 0,Y 272.802,Z 375.642,A -85,B 0,C 180,E1 -18065.807,E2 -18065.807} C_VEL
LIN {X 0,Y 271.923,Z 388.676,A -85,B 0,C 180,E1 -18066.432,E2 -18066.432} C_VEL
LIN {X 0,Y 270.903,Z 400.796,A -85,B 0,C 180,E1 -18067.298,E2 -18067.298} C_VEL
LIN {X 0,Y 269.534,Z 412.209,A -85,B 0,C 180,E1 -18068.387,E2 -18068.387} C_VEL
LIN {X 0,Y 267.907,Z 423.967,A -85,B 0,C 180,E1 -18069.858,E2 -18069.858} C_VEL
LIN {X 0,Y 266.526,Z 434.564,A -85,B 0,C 180,E1 -18071.551,E2 -18071.551} C_VEL
LIN {X 0,Y 265.13,Z 444.069,A -85,B 0,C 180,E1 -18073.441,E2 -18073.441} C_VEL
LIN {X 0,Y 263.638,Z 453.206,A -85,B 0,C 180,E1 -18075.722,E2 -18075.722} C_VEL
LIN {X 0,Y 262.525,Z 460.557,A -85,B 0,C 180,E1 -18078.023,E2 -18078.023} C_VEL
LIN {X 0,Y 261.904,Z 465.518,A -85,B 0,C 180,E1 -18079.953,E2 -18079.953} C_VEL
LIN {X 0,Y 261.373,Z 470.319,A -85,B 0,C 180,E1 -18082.271,E2 -18082.271} C_VEL
LIN {X 0,Y 261.102,Z 474.351,A -85,B 0,C 180,E1 -18084.861,E2 -18084.861} C_VEL
LIN {X 0,Y 261.037,Z 476.605,A -85,B 0,C 180,E1 -18086.911,E2 -18086.911} C_VEL
LIN {X 0,Y 261.047,Z 477.836,A -85,B 0,C 180,E1 -18088.455,E2 -18088.455} C_VEL
LIN {X 0,Y 261.084,Z 478.642,A -85,B 0,C 180,E1 -18089.998,E2 -18089.998} C_VEL
LIN {X 0,Y 261.046,Z 479.023,A -85,B 0,C 180,E1 -18091.54,E2 -18091.54} C_VEL
LIN {X 0,Y 261.082,Z 478.637,A -85,B 0,C 180,E1 -18094.63,E2 -18094.63} C_VEL
LIN {X 0,Y 261.25,Z 477.859,A -85,B 0,C 180,E1 -18096.175,E2 -18096.175} C_VEL
LIN {X 0,Y 261.917,Z 475.042,A -85,B 0,C 180,E1 -18099.262,E2 -18099.262} C_VEL
LIN {X 0,Y 262.778,Z 471.831,A -85,B 0,C 180,E1 -18101.569,E2 -18101.569} C_VEL
LIN {X 0,Y 264.006,Z 467.578,A -85,B 0,C 180,E1 -18103.86,E2 -18103.86} C_VEL
LIN {X 0,Y 266.043,Z 461.17,A -85,B 0,C 180,E1 -18106.495,E2 -18106.495} C_VEL
LIN {X 0,Y 268.225,Z 454.188,A -85,B 0,C 180,E1 -18108.719,E2 -18108.719} C_VEL
LIN {X 0,Y 270.34,Z 446.232,A -85,B 0,C 180,E1 -18110.763,E2 -18110.763} C_VEL
LIN {X 0,Y 272.9,Z 436.641,A -85,B 0,C 180,E1 -18112.721,E2 -18112.721} C_VEL
LIN {X 0,Y 275.569,Z 425.709,A -85,B 0,C 180,E1 -18114.481,E2 -18114.481} C_VEL
LIN {X 0,Y 277.931,Z 414.679,A -85,B 0,C 180,E1 -18115.859,E2 -18115.859} C_VEL
LIN {X 0,Y 280.093,Z 402.369,A -85,B 0,C 180,E1 -18117.048,E2 -18117.048} C_VEL
LIN {X 0,Y 281.868,Z 389.912,A -85,B 0,C 180,E1 -18117.92,E2 -18117.92} C_VEL
LIN {X 0,Y 283.217,Z 376.07,A -85,B 0,C 180,E1 -18118.569,E2 -18118.569} C_VEL
LIN {X 0,Y 284.345,Z 350.174,A -85,B 0,C 180,E1 -18119.281,E2 -18119.281} C_VEL
LIN {X 0,Y 285.771,Z 314.21,A -85,B 0,C 180,E1 -18120.206,E2 -18120.206} C_VEL
LIN {X 0,Y 283.14,Z 299.634,A -85,B 0,C 180,E1 -18121.059,E2 -18121.059} C_VEL
LIN {X 0,Y 276.389,Z 284.915,A -85,B 0,C 180,E1 -18122.608,E2 -18122.608} C_VEL
LIN {X 0,Y 268.717,Z 270.599,A -85,B 0,C 180,E1 -18124.452,E2 -18124.452} C_VEL
LIN {X 0,Y 266.551,Z 266.442,A -85,B 0,C 180,E1 -18125.08,E2 -18125.08} C_VEL
LIN {X 0,Y 265.037,Z 260.922,A -85,B 0,C 180,E1 -18127.578,E2 -18127.578} C_VEL
LIN {X 0,Y 263.141,Z 254.283,A -85,B 0,C 180,E1 -18130.994,E2 -18130.994} C_VEL
LIN {X 0,Y 263.107,Z 254.211,A -85,B 0,C 180,E1 -18133.984,E2 -18133.984} C_VEL
LIN {X 0,Y 263.083,Z 254.204,A -85,B 0,C 180,E1 -18138.413,E2 -18138.413} C_VEL
LIN {X 0,Y 263.149,Z 254.206,A -85,B 0,C 180,E1 -18142.096,E2 -18142.096} C_VEL
LIN {X 0,Y 263.153,Z 254.206,A -85,B 0,C 180,E1 -18145.88,E2 -18145.88} C_VEL
LIN {X 0,Y 263.126,Z 254.208,A -85,B 0,C 180,E1 -18149.498,E2 -18149.498} C_VEL
LIN {X 0,Y 263.136,Z 254.208,A -85,B 0,C 180,E1 -18152.991,E2 -18152.991} C_VEL
LIN {X 0,Y 263.115,Z 254.209,A -85,B 0,C 180,E1 -18156.375,E2 -18156.375} C_VEL
LIN {X 0,Y 263.204,Z 254.19,A -85,B 0,C 180,E1 -18159.683,E2 -18159.683} C_VEL
LIN {X 0,Y 263.304,Z 254.181,A -85,B 0,C 180,E1 -18164.514,E2 -18164.514} C_VEL
LIN {X 0,Y 263.341,Z 254.177,A -85,B 0,C 180,E1 -18169.227,E2 -18169.227} C_VEL
LIN {X 0,Y 263.519,Z 254.145,A -85,B 0,C 180,E1 -18172.331,E2 -18172.331} C_VEL
LIN {X 0,Y 263.723,Z 254.133,A -85,B 0,C 180,E1 -18178.467,E2 -18178.467} C_VEL
LIN {X 0,Y 263.719,Z 254.124,A -85,B 0,C 180,E1 -18181.521,E2 -18181.521} C_VEL
LIN {X 0,Y 263.508,Z 254.163,A -85,B 0,C 180,E1 -18187.657,E2 -18187.657} C_VEL
LIN {X 0,Y 263.331,Z 254.181,A -85,B 0,C 180,E1 -18190.761,E2 -18190.761} C_VEL
LIN {X 0,Y 263.303,Z 254.186,A -85,B 0,C 180,E1 -18195.474,E2 -18195.474} C_VEL
LIN {X 0,Y 263.215,Z 254.193,A -85,B 0,C 180,E1 -18200.303,E2 -18200.303} C_VEL
LIN {X 0,Y 263.168,Z 254.199,A -85,B 0,C 180,E1 -18205.288,E2 -18205.288} C_VEL
LIN {X 0,Y 263.123,Z 254.195,A -85,B 0,C 180,E1 -18209.605,E2 -18209.605} C_VEL
LIN {X 0,Y 263.158,Z 254.475,A -85,B 0,C 180,E1 -18210.484,E2 -18210.484} C_VEL
LIN {X 0,Y 265.051,Z 260.948,A -85,B 0,C 180,E1 -18213.657,E2 -18213.657} C_VEL
LIN {X 0,Y 267.581,Z 265.315,A -85,B 0,C 180,E1 -18214.384,E2 -18214.384} C_VEL
LIN {X 0,Y 275.124,Z 278.612,A -85,B 0,C 180,E1 -18216.2,E2 -18216.2} C_VEL
LIN {X 0,Y 282.194,Z 292.946,A -85,B 0,C 180,E1 -18217.818,E2 -18217.818} C_VEL
LIN {X 0,Y 286.027,Z 302.332,A -85,B 0,C 180,E1 -18218.693,E2 -18218.693} C_VEL
LIN {X 0,Y 285.747,Z 314.998,A -85,B 0,C 180,E1 -18219.051,E2 -18219.051} C_VEL
LIN {X 0,Y 283.386,Z 369.403,A -85,B 0,C 180,E1 -18220.481,E2 -18220.481} C_VEL
LIN {X 0,Y 282.183,Z 382.845,A -85,B 0,C 180,E1 -18221.118,E2 -18221.118} C_VEL
LIN {X 0,Y 280.609,Z 395.045,A -85,B 0,C 180,E1 -18221.971,E2 -18221.971} C_VEL
LIN {X 0,Y 278.735,Z 406.158,A -85,B 0,C 180,E1 -18223.017,E2 -18223.017} C_VEL
LIN {X 0,Y 276.477,Z 417.272,A -85,B 0,C 180,E1 -18224.366,E2 -18224.366} C_VEL
LIN {X 0,Y 274.217,Z 426.969,A -85,B 0,C 180,E1 -18225.848,E2 -18225.848} C_VEL
LIN {X 0,Y 271.607,Z 436.826,A -85,B 0,C 180,E1 -18227.723,E2 -18227.723} C_VEL
LIN {X 0,Y 269.242,Z 445.25,A -85,B 0,C 180,E1 -18229.759,E2 -18229.759} C_VEL
LIN {X 0,Y 266.868,Z 453.177,A -85,B 0,C 180,E1 -18232.178,E2 -18232.178} C_VEL
LIN {X 0,Y 265.138,Z 458.733,A -85,B 0,C 180,E1 -18234.331,E2 -18234.331} C_VEL
LIN {X 0,Y 263.591,Z 463.839,A -85,B 0,C 180,E1 -18236.87,E2 -18236.87} C_VEL
LIN {X 0,Y 262.434,Z 467.581,A -85,B 0,C 180,E1 -18239.418,E2 -18239.418} C_VEL
LIN {X 0,Y 261.434,Z 470.5,A -85,B 0,C 180,E1 -18242.496,E2 -18242.496} C_VEL
LIN {X 0,Y 261.01,Z 471.535,A -85,B 0,C 180,E1 -18244.483,E2 -18244.483} C_VEL
LIN {X 0,Y 260.754,Z 471.909,A -85,B 0,C 180,E1 -18246.384,E2 -18246.384} C_VEL
LIN {X 0,Y 260.667,Z 471.806,A -85,B 0,C 180,E1 -18247.826,E2 -18247.826} C_VEL
LIN {X 0,Y 260.677,Z 470.571,A -85,B 0,C 180,E1 -18250.644,E2 -18250.644} C_VEL
LIN {X 0,Y 260.812,Z 468.773,A -85,B 0,C 180,E1 -18252.76,E2 -18252.76} C_VEL
LIN {X 0,Y 261.284,Z 465.2,A -85,B 0,C 180,E1 -18255.508,E2 -18255.508} C_VEL
LIN {X 0,Y 261.739,Z 461.51,A -85,B 0,C 180,E1 -18257.598,E2 -18257.598} C_VEL
LIN {X 0,Y 262.586,Z 455.047,A -85,B 0,C 180,E1 -18260.373,E2 -18260.373} C_VEL
LIN {X 0,Y 263.577,Z 448.01,A -85,B 0,C 180,E1 -18262.726,E2 -18262.726} C_VEL
LIN {X 0,Y 264.728,Z 440.789,A -85,B 0,C 180,E1 -18264.671,E2 -18264.671} C_VEL
LIN {X 0,Y 266.174,Z 431.062,A -85,B 0,C 180,E1 -18266.786,E2 -18266.786} C_VEL
LIN {X 0,Y 267.927,Z 419.979,A -85,B 0,C 180,E1 -18268.687,E2 -18268.687} C_VEL
LIN {X 0,Y 269.39,Z 408.854,A -85,B 0,C 180,E1 -18270.189,E2 -18270.189} C_VEL
LIN {X 0,Y 270.728,Z 396.388,A -85,B 0,C 180,E1 -18271.49,E2 -18271.49} C_VEL
LIN {X 0,Y 271.835,Z 384.52,A -85,B 0,C 180,E1 -18272.41,E2 -18272.41} C_VEL
LIN {X 0,Y 272.673,Z 371.768,A -85,B 0,C 180,E1 -18273.096,E2 -18273.096} C_VEL
LIN {X 0,Y 273.289,Z 354.156,A -85,B 0,C 180,E1 -18273.642,E2 -18273.642} C_VEL
LIN {X 0,Y 274.794,Z 297.469,A -85,B 0,C 180,E1 -18275.134,E2 -18275.134} C_VEL
LIN {X 0,Y 272.114,Z 281.56,A -85,B 0,C 180,E1 -18275.802,E2 -18275.802} C_VEL
LIN {X 0,Y 264.893,Z 261.01,A -85,B 0,C 180,E1 -18277.058,E2 -18277.058} C_VEL
LIN {X 0,Y 264.297,Z 258.111,A -85,B 0,C 180,E1 -18278.027,E2 -18278.027} C_VEL
LIN {X 0,Y 263.436,Z 254.334,A -85,B 0,C 180,E1 -18279.561,E2 -18279.561} C_VEL
LIN {X 0,Y 263.27,Z 254.19,A -85,B 0,C 180,E1 -18283.904,E2 -18283.904} C_VEL
LIN {X 0,Y 263.225,Z 254.18,A -85,B 0,C 180,E1 -18287.082,E2 -18287.082} C_VEL
LIN {X 0,Y 263.171,Z 254.2,A -85,B 0,C 180,E1 -18290.847,E2 -18290.847} C_VEL
LIN {X 0,Y 263.096,Z 254.211,A -85,B 0,C 180,E1 -18295.305,E2 -18295.305} C_VEL
LIN {X 0,Y 263.098,Z 254.213,A -85,B 0,C 180,E1 -18298.742,E2 -18298.742} C_VEL
LIN {X 0,Y 263.102,Z 254.205,A -85,B 0,C 180,E1 -18302.295,E2 -18302.295} C_VEL
LIN {X 0,Y 263.149,Z 254.204,A -85,B 0,C 180,E1 -18306.766,E2 -18306.766} C_VEL
LIN {X 0,Y 263.069,Z 254.203,A -85,B 0,C 180,E1 -18309.882,E2 -18309.882} C_VEL
LIN {X 0,Y 263.057,Z 254.216,A -85,B 0,C 180,E1 -18314.001,E2 -18314.001} C_VEL
LIN {X 0,Y 263.063,Z 254.203,A -85,B 0,C 180,E1 -18318.425,E2 -18318.425} C_VEL
LIN {X 0,Y 263.125,Z 254.203,A -85,B 0,C 180,E1 -18322.106,E2 -18322.106} C_VEL
LIN {X 0,Y 263.14,Z 254.203,A -85,B 0,C 180,E1 -18325.893,E2 -18325.893} C_VEL
LIN {X 0,Y 263.099,Z 254.19,A -85,B 0,C 180,E1 -18329.508,E2 -18329.508} C_VEL
LIN {X 0,Y 263.104,Z 254.201,A -85,B 0,C 180,E1 -18333.001,E2 -18333.001} C_VEL
LIN {X 0,Y 263.111,Z 254.208,A -85,B 0,C 180,E1 -18336.388,E2 -18336.388} C_VEL
LIN {X 0,Y 263.205,Z 254.191,A -85,B 0,C 180,E1 -18339.696,E2 -18339.696} C_VEL
LIN {X 0,Y 263.31,Z 254.168,A -85,B 0,C 180,E1 -18344.526,E2 -18344.526} C_VEL
LIN {X 0,Y 263.355,Z 254.178,A -85,B 0,C 180,E1 -18349.24,E2 -18349.24} C_VEL
LIN {X 0,Y 263.53,Z 254.152,A -85,B 0,C 180,E1 -18352.343,E2 -18352.343} C_VEL
LIN {X 0,Y 263.736,Z 254.118,A -85,B 0,C 180,E1 -18358.457,E2 -18358.457} C_VEL
LIN {X 0,Y 263.531,Z 254.153,A -85,B 0,C 180,E1 -18359.308,E2 -18359.308} C_VEL
LIN {X 0,Y 262.729,Z 254.26,A -85,B 0,C 180,E1 -18360.147,E2 -18360.147} C_VEL
LIN {X 0,Y 258.738,Z 254.761,A -85,B 0,C 180,E1 -18362.63,E2 -18362.63} C_VEL
LIN {X 0,Y 256.625,Z 255.018,A -85,B 0,C 180,E1 -18364.351,E2 -18364.351} C_VEL
LIN {X 0,Y 256.333,Z 255.048,A -85,B 0,C 180,E1 -18365.241,E2 -18365.241} C_VEL
LIN {X 0,Y 256.467,Z 255.024,A -85,B 0,C 180,E1 -18367.881,E2 -18367.881} C_VEL
LIN {X 0,Y 256.292,Z 255.046,A -85,B 0,C 180,E1 -18371.073,E2 -18371.073} C_VEL
LIN {X 0,Y 256.246,Z 255.064,A -85,B 0,C 180,E1 -18375.924,E2 -18375.924} C_VEL
LIN {X 0,Y 256.14,Z 255.063,A -85,B 0,C 180,E1 -18380.903,E2 -18380.903} C_VEL
LIN {X 0,Y 256.15,Z 255.079,A -85,B 0,C 180,E1 -18385.115,E2 -18385.115} C_VEL
LIN {X 0,Y 256.07,Z 255.075,A -85,B 0,C 180,E1 -18389.611,E2 -18389.611} C_VEL
LIN {X 0,Y 256.085,Z 255.088,A -85,B 0,C 180,E1 -18393.296,E2 -18393.296} C_VEL
LIN {X 0,Y 256.106,Z 255.074,A -85,B 0,C 180,E1 -18397.265,E2 -18397.265} C_VEL
LIN {X 0,Y 256.028,Z 255.092,A -85,B 0,C 180,E1 -18401.215,E2 -18401.215} C_VEL
LIN {X 0,Y 256.037,Z 255.093,A -85,B 0,C 180,E1 -18405.541,E2 -18405.541} C_VEL
LIN {X 0,Y 256.038,Z 255.09,A -85,B 0,C 180,E1 -18408.79,E2 -18408.79} C_VEL
LIN {X 0,Y 256.122,Z 255.077,A -85,B 0,C 180,E1 -18412.863,E2 -18412.863} C_VEL
LIN {X 0,Y 256.17,Z 255.271,A -85,B 0,C 180,E1 -18416.821,E2 -18416.821} C_VEL
LIN {X 0,Y 258.278,Z 265.188,A -85,B 0,C 180,E1 -18420.67,E2 -18420.67} C_VEL
LIN {X 0,Y 258.711,Z 267.404,A -85,B 0,C 180,E1 -18421.383,E2 -18421.383} C_VEL
LIN {X 0,Y 263.864,Z 282.265,A -85,B 0,C 180,E1 -18422.351,E2 -18422.351} C_VEL
LIN {X 0,Y 268.01,Z 311.814,A -85,B 0,C 180,E1 -18423.571,E2 -18423.571} C_VEL
LIN {X 0,Y 266.098,Z 375.642,A -85,B 0,C 180,E1 -18425.313,E2 -18425.313} C_VEL
LIN {X 0,Y 265.165,Z 389.416,A -85,B 0,C 180,E1 -18426.002,E2 -18426.002} C_VEL
LIN {X 0,Y 263.975,Z 402.357,A -85,B 0,C 180,E1 -18426.979,E2 -18426.979} C_VEL
LIN {X 0,Y 262.516,Z 414.154,A -85,B 0,C 180,E1 -18428.192,E2 -18428.192} C_VEL
LIN {X 0,Y 260.831,Z 425.53,A -85,B 0,C 180,E1 -18429.699,E2 -18429.699} C_VEL
LIN {X 0,Y 259.369,Z 436.235,A -85,B 0,C 180,E1 -18431.522,E2 -18431.522} C_VEL
LIN {X 0,Y 257.986,Z 445.018,A -85,B 0,C 180,E1 -18433.377,E2 -18433.377} C_VEL
LIN {X 0,Y 256.504,Z 453.982,A -85,B 0,C 180,E1 -18435.722,E2 -18435.722} C_VEL
LIN {X 0,Y 255.421,Z 461.157,A -85,B 0,C 180,E1 -18438.088,E2 -18438.088} C_VEL
LIN {X 0,Y 254.659,Z 466.859,A -85,B 0,C 180,E1 -18440.466,E2 -18440.466} C_VEL
LIN {X 0,Y 254.189,Z 471.332,A -85,B 0,C 180,E1 -18442.85,E2 -18442.85} C_VEL
LIN {X 0,Y 253.991,Z 474.705,A -85,B 0,C 180,E1 -18445.236,E2 -18445.236} C_VEL
LIN {X 0,Y 253.94,Z 476.374,A -85,B 0,C 180,E1 -18446.825,E2 -18446.825} C_VEL
LIN {X 0,Y 253.957,Z 477.635,A -85,B 0,C 180,E1 -18448.412,E2 -18448.412} C_VEL
LIN {X 0,Y 253.992,Z 478.493,A -85,B 0,C 180,E1 -18449.998,E2 -18449.998} C_VEL
LIN {X 0,Y 253.956,Z 478.91,A -85,B 0,C 180,E1 -18451.583,E2 -18451.583} C_VEL
LIN {X 0,Y 254.009,Z 478.581,A -85,B 0,C 180,E1 -18454.759,E2 -18454.759} C_VEL
LIN {X 0,Y 254.182,Z 477.844,A -85,B 0,C 180,E1 -18456.347,E2 -18456.347} C_VEL
LIN {X 0,Y 254.462,Z 476.682,A -85,B 0,C 180,E1 -18457.935,E2 -18457.935} C_VEL
LIN {X 0,Y 255.467,Z 473.131,A -85,B 0,C 180,E1 -18461.1,E2 -18461.1} C_VEL
LIN {X 0,Y 256.65,Z 469.31,A -85,B 0,C 180,E1 -18463.457,E2 -18463.457} C_VEL
LIN {X 0,Y 258.226,Z 464.393,A -85,B 0,C 180,E1 -18465.79,E2 -18465.79} C_VEL
LIN {X 0,Y 260.341,Z 458.225,A -85,B 0,C 180,E1 -18468.083,E2 -18468.083} C_VEL
LIN {X 0,Y 262.591,Z 450.582,A -85,B 0,C 180,E1 -18470.358,E2 -18470.358} C_VEL
LIN {X 0,Y 265.332,Z 441.025,A -85,B 0,C 180,E1 -18472.583,E2 -18472.583} C_VEL
LIN {X 0,Y 268.1,Z 431.175,A -85,B 0,C 180,E1 -18474.383,E2 -18474.383} C_VEL
LIN {X 0,Y 270.644,Z 420.137,A -85,B 0,C 180,E1 -18475.987,E2 -18475.987} C_VEL
LIN {X 0,Y 272.911,Z 409.35,A -85,B 0,C 180,E1 -18477.197,E2 -18477.197} C_VEL
LIN {X 0,Y 274.898,Z 397.506,A -85,B 0,C 180,E1 -18478.224,E2 -18478.224} C_VEL
LIN {X 0,Y 276.609,Z 384.496,A -85,B 0,C 180,E1 -18479.027,E2 -18479.027} C_VEL
LIN {X 0,Y 277.777,Z 370.861,A -85,B 0,C 180,E1 -18479.551,E2 -18479.551} C_VEL
LIN {X 0,Y 279.975,Z 315.039,A -85,B 0,C 180,E1 -18481.041,E2 -18481.041} C_VEL
LIN {X 0,Y 277.589,Z 302.298,A -85,B 0,C 180,E1 -18481.83,E2 -18481.83} C_VEL
LIN {X 0,Y 271.076,Z 287.953,A -85,B 0,C 180,E1 -18483.414,E2 -18483.414} C_VEL
LIN {X 0,Y 264.016,Z 274.82,A -85,B 0,C 180,E1 -18485.181,E2 -18485.181} C_VEL
LIN {X 0,Y 259.358,Z 266.413,A -85,B 0,C 180,E1 -18486.487,E2 -18486.487} C_VEL
LIN {X 0,Y 257.21,Z 259.061,A -85,B 0,C 180,E1 -18490.08,E2 -18490.08} C_VEL
LIN {X 0,Y 256.054,Z 255.1,A -85,B 0,C 180,E1 -18492.364,E2 -18492.364} C_VEL
LIN {X 0,Y 256.028,Z 255.068,A -85,B 0,C 180,E1 -18496.66,E2 -18496.66} C_VEL
LIN {X 0,Y 256.069,Z 255.082,A -85,B 0,C 180,E1 -18500.851,E2 -18500.851} C_VEL
LIN {X 0,Y 256.123,Z 255.079,A -85,B 0,C 180,E1 -18502.86,E2 -18502.86} C_VEL
LIN {X 0,Y 256.067,Z 255.081,A -85,B 0,C 180,E1 -18506.701,E2 -18506.701} C_VEL
LIN {X 0,Y 256.054,Z 255.082,A -85,B 0,C 180,E1 -18510.387,E2 -18510.387} C_VEL
LIN {X 0,Y 256.077,Z 255.08,A -85,B 0,C 180,E1 -18513.947,E2 -18513.947} C_VEL
LIN {X 0,Y 256.055,Z 255.088,A -85,B 0,C 180,E1 -18517.396,E2 -18517.396} C_VEL
LIN {X 0,Y 256.124,Z 255.08,A -85,B 0,C 180,E1 -18520.769,E2 -18520.769} C_VEL
LIN {X 0,Y 256.224,Z 255.059,A -85,B 0,C 180,E1 -18524.075,E2 -18524.075} C_VEL
LIN {X 0,Y 256.282,Z 255.054,A -85,B 0,C 180,E1 -18528.927,E2 -18528.927} C_VEL
LIN {X 0,Y 256.461,Z 255.025,A -85,B 0,C 180,E1 -18532.119,E2 -18532.119} C_VEL
LIN {X 0,Y 256.432,Z 255.029,A -85,B 0,C 180,E1 -18536.852,E2 -18536.852} C_VEL
LIN {X 0,Y 256.685,Z 255.009,A -85,B 0,C 180,E1 -18538.425,E2 -18538.425} C_VEL
LIN {X 0,Y 256.682,Z 255,A -85,B 0,C 180,E1 -18541.563,E2 -18541.563} C_VEL
LIN {X 0,Y 256.426,Z 255.035,A -85,B 0,C 180,E1 -18546.563,E2 -18546.563} C_VEL
LIN {X 0,Y 256.41,Z 255.036,A -85,B 0,C 180,E1 -18549.459,E2 -18549.459} C_VEL
LIN {X 0,Y 256.217,Z 255.066,A -85,B 0,C 180,E1 -18554.285,E2 -18554.285} C_VEL
LIN {X 0,Y 256.156,Z 255.073,A -85,B 0,C 180,E1 -18557.559,E2 -18557.559} C_VEL
LIN {X 0,Y 256.119,Z 255.083,A -85,B 0,C 180,E1 -18561.105,E2 -18561.105} C_VEL
LIN {X 0,Y 256.146,Z 255.074,A -85,B 0,C 180,E1 -18565.125,E2 -18565.125} C_VEL
LIN {X 0,Y 256.123,Z 255.212,A -85,B 0,C 180,E1 -18569.113,E2 -18569.113} C_VEL
LIN {X 0,Y 257.798,Z 261.084,A -85,B 0,C 180,E1 -18572.195,E2 -18572.195} C_VEL
LIN {X 0,Y 260.141,Z 265.149,A -85,B 0,C 180,E1 -18572.927,E2 -18572.927} C_VEL
LIN {X 0,Y 266.587,Z 275.868,A -85,B 0,C 180,E1 -18574.582,E2 -18574.582} C_VEL
LIN {X 0,Y 273.793,Z 289.533,A -85,B 0,C 180,E1 -18576.347,E2 -18576.347} C_VEL
LIN {X 0,Y 279.575,Z 302.389,A -85,B 0,C 180,E1 -18577.722,E2 -18577.722} C_VEL
LIN {X 0,Y 280.418,Z 304.957,A -85,B 0,C 180,E1 -18577.936,E2 -18577.936} C_VEL
LIN {X 0,Y 277.56,Z 369.127,A -85,B 0,C 180,E1 -18579.64,E2 -18579.64} C_VEL
LIN {X 0,Y 276.298,Z 382.922,A -85,B 0,C 180,E1 -18580.302,E2 -18580.302} C_VEL
LIN {X 0,Y 274.716,Z 394.837,A -85,B 0,C 180,E1 -18581.145,E2 -18581.145} C_VEL
LIN {X 0,Y 272.742,Z 406.065,A -85,B 0,C 180,E1 -18582.209,E2 -18582.209} C_VEL
LIN {X 0,Y 270.403,Z 417.18,A -85,B 0,C 180,E1 -18583.577,E2 -18583.577} C_VEL
LIN {X 0,Y 267.806,Z 427.738,A -85,B 0,C 180,E1 -18585.224,E2 -18585.224} C_VEL
LIN {X 0,Y 265.292,Z 436.79,A -85,B 0,C 180,E1 -18586.991,E2 -18586.991} C_VEL
LIN {X 0,Y 262.793,Z 445.239,A -85,B 0,C 180,E1 -18589.068,E2 -18589.068} C_VEL
LIN {X 0,Y 260.2,Z 453.361,A -85,B 0,C 180,E1 -18591.597,E2 -18591.597} C_VEL
LIN {X 0,Y 258.124,Z 459.726,A -85,B 0,C 180,E1 -18594.174,E2 -18594.174} C_VEL
LIN {X 0,Y 256.523,Z 464.571,A -85,B 0,C 180,E1 -18596.777,E2 -18596.777} C_VEL
LIN {X 0,Y 255.715,Z 467.083,A -85,B 0,C 180,E1 -18598.524,E2 -18598.524} C_VEL
LIN {X 0,Y 255.005,Z 469.051,A -85,B 0,C 180,E1 -18600.262,E2 -18600.262} C_VEL
LIN {X 0,Y 254.446,Z 470.55,A -85,B 0,C 180,E1 -18602.095,E2 -18602.095} C_VEL
LIN {X 0,Y 254.042,Z 471.463,A -85,B 0,C 180,E1 -18603.731,E2 -18603.731} C_VEL
LIN {X 0,Y 253.692,Z 472,A -85,B 0,C 180,E1 -18606.071,E2 -18606.071} C_VEL
LIN {X 0,Y 253.531,Z 471.544,A -85,B 0,C 180,E1 -18608.88,E2 -18608.88} C_VEL
LIN {X 0,Y 253.583,Z 470.647,A -85,B 0,C 180,E1 -18610.578,E2 -18610.578} C_VEL
LIN {X 0,Y 253.676,Z 469.299,A -85,B 0,C 180,E1 -18612.26,E2 -18612.26} C_VEL
LIN {X 0,Y 253.882,Z 467.518,A -85,B 0,C 180,E1 -18613.932,E2 -18613.932} C_VEL
LIN {X 0,Y 254.363,Z 463.916,A -85,B 0,C 180,E1 -18616.42,E2 -18616.42} C_VEL
LIN {X 0,Y 254.963,Z 459.159,A -85,B 0,C 180,E1 -18618.877,E2 -18618.877} C_VEL
LIN {X 0,Y 255.838,Z 452.798,A -85,B 0,C 180,E1 -18621.414,E2 -18621.414} C_VEL
LIN {X 0,Y 256.957,Z 445.509,A -85,B 0,C 180,E1 -18623.722,E2 -18623.722} C_VEL
LIN {X 0,Y 258.265,Z 437.743,A -85,B 0,C 180,E1 -18625.711,E2 -18625.711} C_VEL
LIN {X 0,Y 259.782,Z 428.234,A -85,B 0,C 180,E1 -18627.693,E2 -18627.693} C_VEL
LIN {X 0,Y 261.389,Z 417.762,A -85,B 0,C 180,E1 -18629.425,E2 -18629.425} C_VEL
LIN {X 0,Y 262.922,Z 406.053,A -85,B 0,C 180,E1 -18630.96,E2 -18630.96} C_VEL
LIN {X 0,Y 264.291,Z 393.709,A -85,B 0,C 180,E1 -18632.193,E2 -18632.193} C_VEL
LIN {X 0,Y 265.429,Z 380.681,A -85,B 0,C 180,E1 -18633.133,E2 -18633.133} C_VEL
